KUKA KRL program: MyProgram_060().src

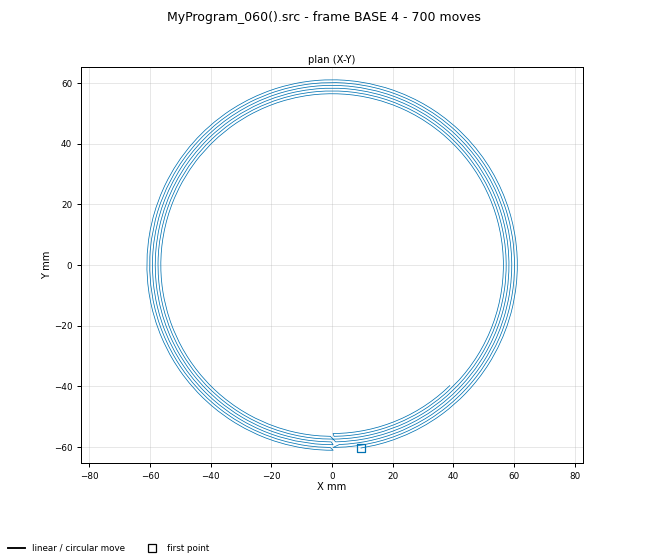
[picture p0: tool path of MyProgram_060().src in frame BASE 4, 700 of 700 moves have a stored position in this frame; points joined in program order, loops and branches not executed]
&ACCESS RVP
&REL 1
&PARAM TEMPLATE = C:\KRC\Roboter\Template\vorgabe
&PARAM EDITMASK = *
DEF MyProgram_060()
; ---- Setting reference (Base) ----
$BASE = BASE_DATA[4]

; --------------------------
; ---- Setting tool (TCP) ----
$TOOL = TOOL_DATA[3]
; --------------------------

$VEL.CP = VEL_APROX_PRINT
Startdeposition()
$VEL.CP = VEL_PRINT
LIN {X 9.5313,Y -60.3261,Z 71,A -85.5574,B 24.8922,C -2.3963,E1 25.0284,E2 529.5228} C_DIS
LIN {X 14.2499,Y -59.3889,Z 71,A -81.7169,B 24.8933,C -2.385,E1 25.0388,E2 525.7139} C_DIS
LIN {X 17.4428,Y -58.5304,Z 71,A -78.0362,B 24.8918,C -2.4016,E1 25.0488,E2 522.0001} C_DIS
LIN {X 20.4744,Y -57.5406,Z 71,A -75.611,B 24.8926,C -2.3923,E1 25.0551,E2 519.6017} C_DIS
LIN {X 24.4545,Y -55.9645,Z 71,A -72.0994,B 24.8931,C -2.3863,E1 25.0642,E2 516.1123} C_DIS
LIN {X 27.8646,Y -54.3472,Z 71,A -68.1205,B 24.8917,C -2.4019,E1 25.0743,E2 512.1067} C_DIS
LIN {X 30.9876,Y -52.6291,Z 71,A -64.3776,B 24.8904,C -2.4171,E1 25.0834,E2 508.339} C_DIS
LIN {X 34.1513,Y -50.6334,Z 71,A -61.0654,B 24.8902,C -2.4192,E1 25.0912,E2 505.0327} C_DIS
LIN {X 36.4572,Y -48.9994,Z 71,A -58.5336,B 24.8899,C -2.4217,E1 25.0969,E2 502.5037} C_DIS
LIN {X 38.3351,Y -47.5447,Z 71,A -55.6589,B 24.8881,C -2.442,E1 25.1032,E2 499.5919} C_DIS
LIN {X 42.1997,Y -44.1508,Z 71,A -51.4902,B 24.8885,C -2.4372,E1 25.1118,E2 495.4512} C_DIS
LIN {X 43.9226,Y -42.4361,Z 71,A -49.1888,B 24.888,C -2.4432,E1 25.1163,E2 493.1454} C_DIS
LIN {X 45.7612,Y -40.4486,Z 71,A -46.6588,B 24.8874,C -2.4493,E1 25.121,E2 490.6124} C_DIS
LIN {X 47.3455,Y -38.5804,Z 71,A -44.3912,B 24.8869,C -2.4545,E1 25.1251,E2 488.3428} C_DIS
LIN {X 49.025,Y -36.4239,Z 71,A -41.5014,B 24.8856,C -2.4692,E1 25.13,E2 485.432} C_DIS
LIN {X 51.0321,Y -33.5526,Z 71,A -38.5025,B 24.8854,C -2.4712,E1 25.1347,E2 482.4432} C_DIS
LIN {X 52.5702,Y -31.0874,Z 71,A -35.4361,B 24.8839,C -2.4873,E1 25.1391,E2 479.3545} C_DIS
LIN {X 54.6001,Y -27.3669,Z 71,A -31.7642,B 24.8835,C -2.4913,E1 25.1439,E2 475.6925} C_DIS
LIN {X 56.3237,Y -23.6157,Z 71,A -27.9982,B 24.8827,C -2.5002,E1 25.1481,E2 471.926} C_DIS
LIN {X 57.7132,Y -19.9822,Z 71,A -23.7879,B 24.8803,C -2.5252,E1 25.1522,E2 467.6801} C_DIS
LIN {X 59.0019,Y -15.7743,Z 71,A -20.3888,B 24.8808,C -2.5199,E1 25.1548,E2 464.3131} C_DIS
LIN {X 59.6127,Y -13.28,Z 71,A -17.5983,B 24.8792,C -2.5369,E1 25.1565,E2 461.4986} C_DIS
LIN {X 60.4839,Y -8.4654,Z 71,A -13.079,B 24.878,C -2.5496,E1 25.1586,E2 456.9758} C_DIS
LIN {X 60.8584,Y -5.1182,Z 71,A -9.9438,B 24.8771,C -2.559,E1 25.1594,E2 453.8369} C_DIS
LIN {X 61.0516,Y -1.6697,Z 71,A -6.9591,B 24.8767,C -2.5628,E1 25.1598,E2 450.8608} C_DIS
LIN {X 61.0519,Y 1.6615,Z 71,A -4.0059,B 24.8762,C -2.5685,E1 25.1597,E2 447.9119} C_DIS
LIN {X 60.9183,Y 4.3667,Z 71,A -0.9984,B 24.8743,C -2.588,E1 25.1591,E2 444.8761} C_DIS
LIN {X 60.5534,Y 7.9589,Z 71,A 2.0459,B 24.8741,C -2.59,E1 25.1582,E2 441.845} C_DIS
LIN {X 60.2672,Y 9.8968,Z 71,A 3.9366,B 24.8734,C -2.597,E1 25.1573,E2 439.9489} C_DIS
LIN {X 59.5946,Y 13.3662,Z 71,A 7.2207,B 24.8725,C -2.6063,E1 25.1554,E2 436.6619} C_DIS
LIN {X 58.852,Y 16.3226,Z 71,A 10.2849,B 24.8711,C -2.62,E1 25.1532,E2 433.5831} C_DIS
LIN {X 57.9096,Y 19.4047,Z 71,A 13.3073,B 24.8702,C -2.6288,E1 25.1506,E2 430.5569} C_DIS
LIN {X 56.5758,Y 23.0049,Z 71,A 16.4909,B 24.8702,C -2.6289,E1 25.1474,E2 427.3908} C_DIS
LIN {X 55.2105,Y 26.1148,Z 71,A 20.5067,B 24.8673,C -2.658,E1 25.1427,E2 423.3278} C_DIS
LIN {X 53.4253,Y 29.5944,Z 71,A 23.4201,B 24.8682,C -2.6495,E1 25.1389,E2 420.4499} C_DIS
LIN {X 51.751,Y 32.4328,Z 71,A 26.9185,B 24.8664,C -2.6673,E1 25.1337,E2 416.9271} C_DIS
LIN {X 49.6974,Y 35.4995,Z 71,A 29.6089,B 24.8674,C -2.6574,E1 25.1295,E2 414.2735} C_DIS
LIN {X 47.4501,Y 38.4518,Z 71,A 33.8937,B 24.8646,C -2.6848,E1 25.122,E2 409.944} C_DIS
LIN {X 44.979,Y 41.3151,Z 71,A 37.3994,B 24.8639,C -2.6916,E1 25.1155,E2 406.4377} C_DIS
LIN {X 42.0159,Y 44.3257,Z 71,A 40.4119,B 24.8654,C -2.6774,E1 25.1096,E2 403.4715} C_DIS
LIN {X 40.4068,Y 45.7971,Z 71,A 42.8829,B 24.864,C -2.6914,E1 25.1044,E2 400.9773} C_DIS
LIN {X 37.3238,Y 48.3424,Z 71,A 46.173,B 24.8644,C -2.6875,E1 25.0973,E2 397.7088} C_DIS
LIN {X 34.8357,Y 50.1649,Z 71,A 49.3042,B 24.8633,C -2.6979,E1 25.0902,E2 394.564} C_DIS
LIN {X 32.4004,Y 51.7711,Z 71,A 52.3355,B 24.8622,C -2.7089,E1 25.0831,E2 391.5166} C_DIS
LIN {X 30.0717,Y 53.1588,Z 71,A 54.7481,B 24.8622,C -2.7094,E1 25.0773,E2 389.1099} C_DIS
LIN {X 27.325,Y 54.6209,Z 71,A 57.7015,B 24.8617,C -2.7139,E1 25.0699,E2 386.154} C_DIS
LIN {X 23.8442,Y 56.2274,Z 71,A 61.6491,B 24.8605,C -2.7258,E1 25.0598,E2 382.1879} C_DIS
LIN {X 20.335,Y 57.5895,Z 71,A 64.8251,B 24.8609,C -2.7211,E1 25.0515,E2 379.0299} C_DIS
LIN {X 17.5465,Y 58.4996,Z 71,A 67.5039,B 24.8609,C -2.7215,E1 25.0444,E2 376.3549} C_DIS
LIN {X 12.2273,Y 59.8376,Z 71,A 72.4673,B 24.861,C -2.7203,E1 25.031,E2 371.4014} C_DIS
LIN {X 7.8287,Y 60.5703,Z 71,A 76.8844,B 24.8604,C -2.7266,E1 25.0187,E2 366.9737} C_DIS
LIN {X 4.1966,Y 60.9298,Z 71,A 80.4406,B 24.8601,C -2.7296,E1 25.0088,E2 363.4121} C_DIS
LIN {X 1.5588,Y 61.055,Z 71,A 83.8521,B 24.858,C -2.7493,E1 24.9992,E2 359.9544} C_DIS
LIN {X -2.3408,Y 61.0299,Z 71,A 86.0215,B 24.8614,C -2.7168,E1 24.9933,E2 357.8622} C_DIS
LIN {X -4.5003,Y 60.9082,Z 71,A 88.4038,B 24.8607,C -2.7234,E1 24.9866,E2 355.4635} C_DIS
LIN {X -7.1884,Y 60.6497,Z 71,A 90.9106,B 24.8609,C -2.7215,E1 24.9797,E2 352.9596} C_DIS
LIN {X -9.8136,Y 60.2811,Z 71,A 93.7308,B 24.8604,C -2.7267,E1 24.9719,E2 350.1247} C_DIS
LIN {X -12.1519,Y 59.8531,Z 71,A 96.1882,B 24.8601,C -2.7295,E1 24.9651,E2 347.6576} C_DIS
LIN {X -16.0091,Y 58.9386,Z 71,A 99.3972,B 24.8615,C -2.7155,E1 24.9565,E2 344.4773} C_DIS
LIN {X -18.5062,Y 58.203,Z 71,A 101.8781,B 24.8617,C -2.7136,E1 24.9499,E2 341.9967} C_DIS
LIN {X -21.2409,Y 57.2618,Z 71,A 104.8189,B 24.8616,C -2.7148,E1 24.9421,E2 339.0473} C_DIS
LIN {X -24.891,Y 55.7722,Z 71,A 108.3276,B 24.8625,C -2.7058,E1 24.9332,E2 335.5519} C_DIS
LIN {X -27.9296,Y 54.314,Z 71,A 111.689,B 24.8626,C -2.7047,E1 24.9247,E2 332.1842} C_DIS
LIN {X -31.0887,Y 52.5694,Z 71,A 114.4199,B 24.8645,C -2.6861,E1 24.9182,E2 329.4896} C_DIS
LIN {X -33.5476,Y 51.0353,Z 71,A 117.4155,B 24.8645,C -2.6864,E1 24.9111,E2 326.4838} C_DIS
LIN {X -35.2032,Y 49.9088,Z 71,A 119.7238,B 24.864,C -2.691,E1 24.9058,E2 324.1566} C_DIS
LIN {X -38.7067,Y 47.2435,Z 71,A 123.6795,B 24.8652,C -2.679,E1 24.8971,E2 320.2151} C_DIS
LIN {X -41.8199,Y 44.5094,Z 71,A 127.6927,B 24.8659,C -2.6726,E1 24.8888,E2 316.201} C_DIS
LIN {X -44.4407,Y 41.8923,Z 71,A 131.5933,B 24.8659,C -2.6723,E1 24.8812,E2 312.2843} C_DIS
LIN {X -47.0833,Y 38.9004,Z 71,A 135.1961,B 24.8671,C -2.6601,E1 24.8747,E2 308.6942} C_DIS
LIN {X -49.9457,Y 35.1511,Z 71,A 138.9483,B 24.8695,C -2.6358,E1 24.8685,E2 304.9819} C_DIS
LIN {X -52.1565,Y 31.7765,Z 71,A 142.9291,B 24.8702,C -2.629,E1 24.8625,E2 300.9973} C_DIS
LIN {X -54.0948,Y 28.3504,Z 71,A 146.6636,B 24.8712,C -2.6192,E1 24.8575,E2 297.2666} C_DIS
LIN {X -55.2292,Y 26.0746,Z 71,A 148.9802,B 24.872,C -2.6109,E1 24.8546,E2 294.9573} C_DIS
LIN {X -56.5378,Y 23.0984,Z 71,A 152.6229,B 24.8718,C -2.6127,E1 24.8506,E2 291.2902} C_DIS
LIN {X -58.0535,Y 18.9702,Z 71,A 156.411,B 24.8737,C -2.594,E1 24.8472,E2 287.5253} C_DIS
LIN {X -59.019,Y 15.7117,Z 71,A 159.9204,B 24.8741,C -2.59,E1 24.8445,E2 284.0052} C_DIS
LIN {X -59.9673,Y 11.5748,Z 71,A 164.0224,B 24.8751,C -2.5797,E1 24.8421,E2 279.9035} C_DIS
LIN {X -60.5089,Y 8.2947,Z 71,A 166.6181,B 24.8769,C -2.5603,E1 24.8411,E2 277.3386} C_DIS
LIN {X -60.9649,Y 3.6625,Z 71,A 170.8735,B 24.8785,C -2.5445,E1 24.84,E2 273.0955} C_DIS
LIN {X -61.0554,Y -1.5469,Z 71,A 176.0124,B 24.8795,C -2.5336,E1 24.8399,E2 267.9518} C_DIS
LIN {X -60.7658,Y -6.133,Z 71,A -179.9583,B 24.8813,C -2.5149,E1 24.8407,E2 263.9428} C_DIS
LIN {X -60.3491,Y -9.3826,Z 71,A -175.9941,B 24.8806,C -2.5217,E1 24.8422,E2 259.9388} C_DIS
LIN {X -59.747,Y -12.6645,Z 71,A -173.4662,B 24.8826,C -2.5011,E1 24.8436,E2 257.4453} C_DIS
LIN {X -59.1871,Y -15.065,Z 71,A -170.4431,B 24.882,C -2.5072,E1 24.8456,E2 254.3899} C_DIS
LIN {X -58.0142,Y -19.0915,Z 71,A -166.5799,B 24.8832,C -2.4943,E1 24.8489,E2 250.5354} C_DIS
LIN {X -56.7141,Y -22.6646,Z 71,A -163.1855,B 24.8845,C -2.4808,E1 24.8523,E2 247.1541} C_DIS
LIN {X -55.5425,Y -25.4007,Z 71,A -160.3729,B 24.8852,C -2.4734,E1 24.8555,E2 244.3438} C_DIS
LIN {X -53.531,Y -29.4038,Z 71,A -156.4605,B 24.8867,C -2.4566,E1 24.8605,E2 240.4507} C_DIS
LIN {X -52.1052,Y -31.8609,Z 71,A -153.6626,B 24.8871,C -2.4522,E1 24.8645,E2 237.6489} C_DIS
LIN {X -50.2298,Y -34.7424,Z 71,A -150.4202,B 24.8879,C -2.4444,E1 24.8695,E2 234.4088} C_DIS
LIN {X -49.0978,Y -36.3255,Z 71,A -147.7959,B 24.8869,C -2.4553,E1 24.874,E2 231.7457} C_DIS
LIN {X -47.1038,Y -38.8757,Z 71,A -145.7362,B 24.8892,C -2.4295,E1 24.8775,E2 229.7381} C_DIS
LIN {X -44.3514,Y -41.9886,Z 71,A -141.8795,B 24.8901,C -2.4201,E1 24.8847,E2 225.8867} C_DIS
LIN {X -42.4737,Y -43.8866,Z 71,A -139.3874,B 24.8906,C -2.4147,E1 24.8896,E2 223.3971} C_DIS
LIN {X -40.1119,Y -46.0553,Z 71,A -136.1393,B 24.8906,C -2.4135,E1 24.8964,E2 220.1388} C_DIS
LIN {X -37.6052,Y -48.1241,Z 71,A -132.9342,B 24.8909,C -2.411,E1 24.9033,E2 216.9274} C_DIS
LIN {X -34.1663,Y -50.6233,Z 71,A -129.0128,B 24.8916,C -2.4032,E1 24.9123,E2 213.0113} C_DIS
LIN {X -31.9807,Y -52.0325,Z 71,A -126.2783,B 24.8914,C -2.4055,E1 24.9188,E2 210.2627} C_DIS
LIN {X -28.8608,Y -53.8255,Z 71,A -122.7562,B 24.8915,C -2.404,E1 24.9274,E2 206.7341} C_DIS
LIN {X -24.5436,Y -55.9257,Z 71,A -118.7195,B 24.8929,C -2.3893,E1 24.9376,E2 202.7222} C_DIS
LIN {X -21.8949,Y -57.0142,Z 71,A -116.0165,B 24.8931,C -2.3871,E1 24.9446,E2 200.0187} C_DIS
LIN {X -19.0924,Y -58.014,Z 71,A -112.065,B 24.8911,C -2.4093,E1 24.9552,E2 196.007} C_DIS
LIN {X -15.3082,Y -59.1246,Z 71,A -110.0337,B 24.8944,C -2.3718,E1 24.9605,E2 194.0618} C_DIS
LIN {X -11.3347,Y -60.0135,Z 71,A -105.6294,B 24.8935,C -2.3823,E1 24.9726,E2 189.6269} C_DIS
LIN {X -8.9195,Y -60.4202,Z 71,A -102.8059,B 24.8925,C -2.3931,E1 24.9804,E2 186.7755} C_DIS
LIN {X -5.3261,Y -60.8421,Z 71,A -100.1582,B 24.894,C -2.3766,E1 24.9877,E2 184.1654} C_DIS
LIN {X -1.8193,Y -61.047,Z 71,A -96.6621,B 24.8936,C -2.3812,E1 24.9975,E2 180.6574} C_DIS
LIN {X 0.3504,Y -61.0663,Z 71,A -94.3682,B 24.893,C -2.3875,E1 25.0039,E2 178.3488} C_DIS
Enddeposition()
LIN {X 0.3504,Y -61.0663,Z 71,A -94.3682,B 24.893,C -2.3875,E1 25.0039,E2 178.3488} C_DIS
Startdeposition()
$VEL.CP = VEL_PRINT
LIN {X -0.6024,Y -60.1527,Z 71,A -97.3329,B 24.8956,C -2.3591,E1 24.9955,E2 181.381} C_DIS
LIN {X -4.5861,Y -59.9805,Z 71,A -100.7162,B 24.8948,C -2.3675,E1 24.9861,E2 184.7453} C_DIS
LIN {X -7.8091,Y -59.6461,Z 71,A -103.721,B 24.8946,C -2.3697,E1 24.9777,E2 187.747} C_DIS
LIN {X -10.2074,Y -59.2836,Z 71,A -106.4784,B 24.8954,C -2.3612,E1 24.9701,E2 190.5271} C_DIS
LIN {X -14.9728,Y -58.262,Z 71,A -111.6213,B 24.8961,C -2.3536,E1 24.9561,E2 195.6951} C_DIS
LIN {X -18.2838,Y -57.3098,Z 71,A -114.2777,B 24.8948,C -2.3683,E1 24.9491,E2 198.3211} C_DIS
LIN {X -22.1363,Y -55.9344,Z 71,A -118.2942,B 24.8946,C -2.3695,E1 24.9385,E2 202.3432} C_DIS
LIN {X -25.8621,Y -54.3125,Z 71,A -121.9851,B 24.894,C -2.3773,E1 24.9292,E2 206.0246} C_DIS
LIN {X -28.523,Y -52.9634,Z 71,A -124.9156,B 24.8938,C -2.3791,E1 24.9219,E2 208.9587} C_DIS
LIN {X -32.2792,Y -50.7619,Z 71,A -128.3777,B 24.8921,C -2.3983,E1 24.9137,E2 212.3858} C_DIS
LIN {X -35.6023,Y -48.4885,Z 71,A -132.4546,B 24.8919,C -2.3999,E1 24.9044,E2 216.4728} C_DIS
LIN {X -37.3846,Y -47.128,Z 71,A -134.7657,B 24.8919,C -2.4003,E1 24.8993,E2 218.7913} C_DIS
LIN {X -39.1876,Y -45.6403,Z 71,A -137.4375,B 24.8923,C -2.3961,E1 24.8935,E2 221.4834} C_DIS
LIN {X -41.213,Y -43.8194,Z 71,A -139.9645,B 24.8917,C -2.4025,E1 24.8884,E2 224.0055} C_DIS
LIN {X -43.7788,Y -41.2562,Z 71,A -143.9978,B 24.892,C -2.3993,E1 24.8805,E2 228.064} C_DIS
LIN {X -46.0507,Y -38.7051,Z 71,A -146.008,B 24.8892,C -2.4293,E1 24.877,E2 230.0116} C_DIS
LIN {X -48.4635,Y -35.6364,Z 71,A -150.0555,B 24.889,C -2.4321,E1 24.8701,E2 234.0718} C_DIS
LIN {X -50.0061,Y -33.4377,Z 71,A -152.5742,B 24.8883,C -2.4391,E1 24.8661,E2 236.5861} C_DIS
LIN {X -51.3259,Y -31.374,Z 71,A -155.0698,B 24.8881,C -2.4421,E1 24.8624,E2 239.0872} C_DIS
LIN {X -52.4055,Y -29.5358,Z 71,A -156.947,B 24.8873,C -2.4502,E1 24.8598,E2 240.9548} C_DIS
LIN {X -53.8809,Y -26.7487,Z 71,A -160.2346,B 24.887,C -2.4533,E1 24.8556,E2 244.2528} C_DIS
LIN {X -55.2221,Y -23.8581,Z 71,A -163.2733,B 24.8863,C -2.4617,E1 24.8521,E2 247.288} C_DIS
LIN {X -56.306,Y -21.1733,Z 71,A -166.1679,B 24.8858,C -2.4672,E1 24.8492,E2 250.1857} C_DIS
LIN {X -57.2806,Y -18.3741,Z 71,A -168.5005,B 24.8842,C -2.4841,E1 24.8471,E2 252.4913} C_DIS
LIN {X -58.3236,Y -14.7331,Z 71,A -171.8693,B 24.8828,C -2.499,E1 24.8446,E2 255.8439} C_DIS
LIN {X -59.0185,Y -11.6424,Z 71,A -175.8143,B 24.8834,C -2.492,E1 24.8423,E2 259.8291} C_DIS
LIN {X -59.7898,Y -6.6302,Z 71,A 179.6959,B 24.8815,C -2.5128,E1 24.8406,E2 264.2958} C_DIS
LIN {X -60.1279,Y -1.812,Z 71,A 175.3491,B 24.8797,C -2.5317,E1 24.8398,E2 268.6237} C_DIS
LIN {X -60.0961,Y 2.6668,Z 71,A 171.1828,B 24.8782,C -2.5469,E1 24.84,E2 272.7787} C_DIS
LIN {X -59.9771,Y 4.6287,Z 71,A 168.4056,B 24.8792,C -2.5371,E1 24.8405,E2 275.5959} C_DIS
LIN {X -59.5679,Y 8.3859,Z 71,A 164.4883,B 24.8786,C -2.543,E1 24.842,E2 279.5225} C_DIS
LIN {X -58.2854,Y 14.882,Z 71,A 159.1838,B 24.875,C -2.5801,E1 24.845,E2 284.7697} C_DIS
LIN {X -57.5897,Y 17.3797,Z 71,A 156.2187,B 24.8751,C -2.5791,E1 24.8474,E2 287.7543} C_DIS
LIN {X -56.6004,Y 20.3742,Z 71,A 152.7791,B 24.875,C -2.5807,E1 24.8506,E2 291.2096} C_DIS
LIN {X -54.5804,Y 25.2911,Z 71,A 147.6942,B 24.8735,C -2.5954,E1 24.8562,E2 296.2874} C_DIS
LIN {X -52.0908,Y 30.0868,Z 71,A 142.7359,B 24.8718,C -2.6134,E1 24.8628,E2 301.2288} C_DIS
LIN {X -50.0697,Y 33.3421,Z 71,A 139.4301,B 24.8702,C -2.6295,E1 24.8678,E2 304.5128} C_DIS
LIN {X -47.9265,Y 36.3542,Z 71,A 135.292,B 24.8703,C -2.628,E1 24.8747,E2 308.6745} C_DIS
LIN {X -45.189,Y 39.7069,Z 71,A 131.43,B 24.8688,C -2.643,E1 24.8816,E2 312.5182} C_DIS
LIN {X -42.5715,Y 42.502,Z 71,A 127.6514,B 24.8682,C -2.6494,E1 24.889,E2 316.2978} C_DIS
LIN {X -38.7988,Y 45.9716,Z 71,A 123.5322,B 24.8657,C -2.6743,E1 24.8975,E2 320.3741} C_DIS
LIN {X -36.4037,Y 47.8889,Z 71,A 119.9369,B 24.8663,C -2.6681,E1 24.9054,E2 323.9974} C_DIS
LIN {X -33.3449,Y 50.0673,Z 71,A 116.4337,B 24.8655,C -2.6764,E1 24.9135,E2 327.4926} C_DIS
LIN {X -30.3333,Y 51.9485,Z 71,A 112.1211,B 24.8666,C -2.6653,E1 24.9239,E2 331.8448} C_DIS
LIN {X -26.9443,Y 53.7838,Z 71,A 109.5322,B 24.864,C -2.6913,E1 24.9302,E2 334.3787} C_DIS
LIN {X -25.1235,Y 54.6584,Z 71,A 107.0936,B 24.8647,C -2.6845,E1 24.9365,E2 336.8395} C_DIS
LIN {X -20.6035,Y 56.5168,Z 71,A 103.1848,B 24.8626,C -2.705,E1 24.9465,E2 340.7081} C_DIS
LIN {X -18.7117,Y 57.1712,Z 71,A 100.3683,B 24.8641,C -2.6897,E1 24.9541,E2 343.5661} C_DIS
LIN {X -15.3925,Y 58.1534,Z 71,A 96.9099,B 24.8641,C -2.6899,E1 24.9634,E2 347.0292} C_DIS
LIN {X -12.2651,Y 58.8918,Z 71,A 94.9035,B 24.8618,C -2.7131,E1 24.9687,E2 348.9829} C_DIS
LIN {X -8.8298,Y 59.5035,Z 71,A 91.5704,B 24.8615,C -2.7153,E1 24.9779,E2 352.314} C_DIS
LIN {X -6.9747,Y 59.7495,Z 71,A 89.4695,B 24.8621,C -2.71,E1 24.9838,E2 354.4291} C_DIS
LIN {X -3.534,Y 60.0517,Z 71,A 86.5713,B 24.8611,C -2.7193,E1 24.9918,E2 357.3064} C_DIS
LIN {X 1.304,Y 60.1414,Z 71,A 82.0334,B 24.8609,C -2.7218,E1 25.0045,E2 361.8384} C_DIS
LIN {X 4.0722,Y 60.0172,Z 71,A 78.6283,B 24.8625,C -2.7062,E1 25.014,E2 365.2794} C_DIS
LIN {X 7.8042,Y 59.6465,Z 71,A 75.1627,B 24.8623,C -2.7077,E1 25.0236,E2 368.7387} C_DIS
LIN {X 12.0069,Y 58.9448,Z 71,A 70.4446,B 24.8639,C -2.6925,E1 25.0366,E2 373.4877} C_DIS
LIN {X 15.4197,Y 58.146,Z 71,A 67.8014,B 24.8626,C -2.705,E1 25.0437,E2 376.097} C_DIS
LIN {X 19.1131,Y 57.0381,Z 71,A 64.5218,B 24.862,C -2.7106,E1 25.0524,E2 379.3574} C_DIS
LIN {X 21.3935,Y 56.2226,Z 71,A 61.8822,B 24.863,C -2.7014,E1 25.0593,E2 382.0134} C_DIS
LIN {X 24.6497,Y 54.873,Z 71,A 58.9077,B 24.8625,C -2.7061,E1 25.0669,E2 384.9696} C_DIS
LIN {X 27.2605,Y 53.624,Z 71,A 55.6988,B 24.8638,C -2.6929,E1 25.075,E2 388.2013} C_DIS
LIN {X 29.7238,Y 52.2994,Z 71,A 53.3009,B 24.8636,C -2.695,E1 25.0808,E2 390.587} C_DIS
LIN {X 33.2527,Y 50.1292,Z 71,A 49.2867,B 24.8644,C -2.6875,E1 25.0903,E2 394.606} C_DIS
LIN {X 36.2291,Y 48.022,Z 71,A 46.3877,B 24.8637,C -2.6945,E1 25.0968,E2 397.4782} C_DIS
LIN {X 38.8634,Y 45.9165,Z 71,A 42.5979,B 24.8656,C -2.6756,E1 25.1051,E2 401.2986} C_DIS
LIN {X 40.7623,Y 44.2392,Z 71,A 40.4405,B 24.8655,C -2.6767,E1 25.1096,E2 403.4448} C_DIS
LIN {X 43.3467,Y 41.7099,Z 71,A 36.8774,B 24.8665,C -2.6668,E1 25.1166,E2 407.0163} C_DIS
LIN {X 44.7731,Y 40.1749,Z 71,A 34.1484,B 24.8686,C -2.6457,E1 25.1218,E2 409.783} C_DIS
LIN {X 48.2371,Y 35.9425,Z 71,A 29.7537,B 24.8679,C -2.6521,E1 25.1293,E2 414.142} C_DIS
LIN {X 50.1978,Y 33.1486,Z 71,A 26.3954,B 24.869,C -2.6415,E1 25.1346,E2 417.5087} C_DIS
LIN {X 51.4362,Y 31.1925,Z 71,A 24.2678,B 24.8694,C -2.6376,E1 25.1377,E2 419.6348} C_DIS
LIN {X 52.9238,Y 28.5959,Z 71,A 21.7482,B 24.8694,C -2.6377,E1 25.1411,E2 422.1409} C_DIS
LIN {X 54.4607,Y 25.5483,Z 71,A 18.7154,B 24.8697,C -2.634,E1 25.1449,E2 425.1664} C_DIS
LIN {X 55.7019,Y 22.7144,Z 71,A 14.5086,B 24.8735,C -2.5961,E1 25.1495,E2 429.4397} C_DIS
LIN {X 56.8361,Y 19.7069,Z 71,A 12.565,B 24.8718,C -2.6135,E1 25.1513,E2 431.3313} C_DIS
LIN {X 57.558,Y 17.4882,Z 71,A 9.0058,B 24.8755,C -2.5754,E1 25.1543,E2 434.9602} C_DIS
LIN {X 58.5266,Y 13.9009,Z 71,A 6.6587,B 24.8738,C -2.5928,E1 25.1558,E2 437.2525} C_DIS
LIN {X 59.4677,Y 9.0697,Z 71,A 2.1525,B 24.8748,C -2.5828,E1 25.1581,E2 441.7561} C_DIS
LIN {X 59.7772,Y 6.7379,Z 71,A -0.8146,B 24.8771,C -2.5585,E1 25.1591,E2 444.7632} C_DIS
LIN {X 60.1241,Y 1.9359,Z 71,A -5.3772,B 24.8784,C -2.5447,E1 25.1598,E2 449.3313} C_DIS
LIN {X 60.1423,Y -1.2551,Z 71,A -7.9162,B 24.8782,C -2.547,E1 25.1597,E2 451.8497} C_DIS
LIN {X 59.9587,Y -4.8584,Z 71,A -11.4456,B 24.8795,C -2.5339,E1 25.1591,E2 455.3892} C_DIS
LIN {X 59.6595,Y -7.707,Z 71,A -13.9397,B 24.8798,C -2.5309,E1 25.1583,E2 457.8756} C_DIS
LIN {X 59.1993,Y -10.6817,Z 71,A -16.9157,B 24.8809,C -2.5192,E1 25.1569,E2 460.8617} C_DIS
LIN {X 58.41,Y -14.3854,Z 71,A -20.7632,B 24.8825,C -2.5022,E1 25.1545,E2 464.7271} C_DIS
LIN {X 57.5402,Y -17.5459,Z 71,A -23.9267,B 24.8835,C -2.4915,E1 25.152,E2 467.8977} C_DIS
LIN {X 56.1297,Y -21.6368,Z 71,A -27.5493,B 24.8835,C -2.4909,E1 25.1486,E2 471.5016} C_DIS
LIN {X 55.2437,Y -23.8085,Z 71,A -29.912,B 24.8845,C -2.4811,E1 25.146,E2 473.8744} C_DIS
LIN {X 53.949,Y -26.6115,Z 71,A -32.8209,B 24.8852,C -2.4732,E1 25.1425,E2 476.7863} C_DIS
LIN {X 51.7218,Y -30.7168,Z 71,A -36.5119,B 24.8847,C -2.4785,E1 25.1376,E2 480.4456} C_DIS
LIN {X 49.2068,Y -34.6039,Z 71,A -41.5992,B 24.8873,C -2.4502,E1 25.1298,E2 485.5744} C_DIS
LIN {X 47.3592,Y -37.0921,Z 71,A -44.6534,B 24.8883,C -2.4399,E1 25.1246,E2 488.6382} C_DIS
LIN {X 45.7436,Y -39.0663,Z 71,A -46.7003,B 24.888,C -2.4427,E1 25.1209,E2 490.6693} C_DIS
LIN {X 44.4188,Y -40.5665,Z 71,A -48.6586,B 24.8886,C -2.4367,E1 25.1173,E2 492.6331} C_DIS
LIN {X 42.6589,Y -42.4135,Z 71,A -51.3079,B 24.8896,C -2.4257,E1 25.1121,E2 495.297} C_DIS
LIN {X 40.0318,Y -44.9012,Z 71,A -54.5017,B 24.8898,C -2.4236,E1 25.1056,E2 498.4828} C_DIS
LIN {X 37.682,Y -46.8912,Z 71,A -57.3654,B 24.8902,C -2.4187,E1 25.0994,E2 501.347} C_DIS
LIN {X 36.2809,Y -47.9831,Z 71,A -59.4249,B 24.8913,C -2.4067,E1 25.0948,E2 503.4273} C_DIS
LIN {X 33.4816,Y -49.9772,Z 71,A -62.5144,B 24.8915,C -2.4044,E1 25.0877,E2 506.5117} C_DIS
LIN {X 30.9995,Y -51.5535,Z 71,A -65.451,B 24.8923,C -2.3961,E1 25.0807,E2 509.4587} C_DIS
LIN {X 28.3987,Y -53.0308,Z 71,A -68.5489,B 24.8932,C -2.3856,E1 25.0731,E2 512.5725} C_DIS
LIN {X 25.2337,Y -54.6071,Z 71,A -71.4802,B 24.8928,C -2.3901,E1 25.0658,E2 515.4855} C_DIS
LIN {X 22.8346,Y -55.653,Z 71,A -73.9642,B 24.8931,C -2.3867,E1 25.0594,E2 517.9717} C_DIS
LIN {X 20.2552,Y -56.6435,Z 71,A -76.6449,B 24.8935,C -2.3821,E1 25.0523,E2 520.6575} C_DIS
LIN {X 17.1851,Y -57.6483,Z 71,A -79.9352,B 24.8943,C -2.3739,E1 25.0435,E2 523.9614} C_DIS
LIN {X 14.4605,Y -58.3917,Z 71,A -82.1861,B 24.8936,C -2.3808,E1 25.0375,E2 526.1925} C_DIS
LIN {X 10.6878,Y -59.1982,Z 71,A -85.6372,B 24.8935,C -2.3824,E1 25.0281,E2 529.6353} C_DIS
LIN {X 8.7278,Y -59.5193,Z 71,A -89.2244,B 24.8968,C -2.3449,E1 25.018,E2 533.3083} C_DIS
LIN {X 4.5328,Y -59.9848,Z 71,A -92.1184,B 24.8949,C -2.3666,E1 25.0101,E2 536.1492} C_DIS
LIN {X 0.3297,Y -60.1458,Z 71,A -94.3994,B 24.8917,C -2.4023,E1 25.004,E2 538.3448} C_DIS
Enddeposition()
LIN {X 0.3297,Y -60.1458,Z 71,A -94.3994,B 24.8917,C -2.4023,E1 25.004,E2 538.3448} C_DIS
Startdeposition()
$VEL.CP = VEL_PRINT
LIN {X 2.3476,Y -59.1901,Z 71,A -92.6158,B 24.8906,C -2.4149,E1 25.009,E2 536.5318} C_DIS
LIN {X 5.1105,Y -59.0155,Z 71,A -89.1553,B 24.8889,C -2.4331,E1 25.0187,E2 533.0299} C_DIS
LIN {X 8.5308,Y -58.6192,Z 71,A -86.7615,B 24.8906,C -2.4149,E1 25.0252,E2 530.6814} C_DIS
LIN {X 10.9463,Y -58.2167,Z 71,A -84.5732,B 24.8907,C -2.4128,E1 25.0312,E2 528.5004} C_DIS
LIN {X 12.903,Y -57.8147,Z 71,A -82.4491,B 24.8902,C -2.4188,E1 25.037,E2 526.3651} C_DIS
LIN {X 15.513,Y -57.169,Z 71,A -79.8384,B 24.8899,C -2.4216,E1 25.0441,E2 523.7516} C_DIS
LIN {X 18.3053,Y -56.3371,Z 71,A -76.8889,B 24.8894,C -2.4278,E1 25.052,E2 520.7927} C_DIS
LIN {X 21.8293,Y -55.0678,Z 71,A -73.7259,B 24.8899,C -2.4223,E1 25.0602,E2 517.6495} C_DIS
LIN {X 23.4437,Y -54.4004,Z 71,A -71.2991,B 24.8881,C -2.4414,E1 25.0665,E2 515.1833} C_DIS
LIN {X 27.932,Y -52.2383,Z 71,A -67.1599,B 24.8888,C -2.4337,E1 25.0768,E2 511.0734} C_DIS
LIN {X 30.5511,Y -50.7507,Z 71,A -63.7965,B 24.8874,C -2.4492,E1 25.085,E2 507.6836} C_DIS
LIN {X 32.8108,Y -49.3199,Z 71,A -61.176,B 24.8869,C -2.455,E1 25.0911,E2 505.0582} C_DIS
LIN {X 36.1038,Y -46.9623,Z 71,A -57.7367,B 24.8872,C -2.452,E1 25.0988,E2 501.6382} C_DIS
LIN {X 38.0627,Y -45.3895,Z 71,A -54.7261,B 24.8854,C -2.4708,E1 25.1053,E2 498.5946} C_DIS
LIN {X 40.9142,Y -42.8374,Z 71,A -51.2565,B 24.8851,C -2.4739,E1 25.1124,E2 495.1317} C_DIS
LIN {X 43.5568,Y -40.1468,Z 71,A -47.873,B 24.8849,C -2.4766,E1 25.1189,E2 491.7565} C_DIS
LIN {X 45.297,Y -38.172,Z 71,A -45.0831,B 24.8837,C -2.4889,E1 25.124,E2 488.9502} C_DIS
LIN {X 47.7459,Y -35.0611,Z 71,A -41.788,B 24.884,C -2.4863,E1 25.1296,E2 485.6768} C_DIS
LIN {X 49.4078,Y -32.6776,Z 71,A -38.2296,B 24.8816,C -2.5118,E1 25.1352,E2 482.0757} C_DIS
LIN {X 50.999,Y -30.1338,Z 71,A -35.3369,B 24.8808,C -2.5198,E1 25.1394,E2 479.1789} C_DIS
LIN {X 53.2383,Y -25.9758,Z 71,A -31.4083,B 24.881,C -2.5177,E1 25.1444,E2 475.2761} C_DIS
LIN {X 54.1566,Y -24.0026,Z 71,A -29.0597,B 24.8799,C -2.5298,E1 25.1471,E2 472.9116} C_DIS
LIN {X 55.3963,Y -20.9808,Z 71,A -25.9604,B 24.8791,C -2.5379,E1 25.1503,E2 469.8104} C_DIS
LIN {X 56.5244,Y -17.7192,Z 71,A -22.9217,B 24.8788,C -2.541,E1 25.1529,E2 466.7817} C_DIS
LIN {X 57.1128,Y -15.721,Z 71,A -20.2553,B 24.8767,C -2.5629,E1 25.1549,E2 464.0787} C_DIS
LIN {X 58.027,Y -11.9084,Z 71,A -16.941,B 24.8767,C -2.5632,E1 25.1569,E2 460.7828} C_DIS
LIN {X 58.4563,Y -9.5834,Z 71,A -13.9915,B 24.8744,C -2.5865,E1 25.1583,E2 457.7957} C_DIS
LIN {X 58.95,Y -5.8274,Z 71,A -11.2766,B 24.8755,C -2.5751,E1 25.1591,E2 455.1237} C_DIS
LIN {X 59.1986,Y -2.139,Z 71,A -7.8773,B 24.8748,C -2.5821,E1 25.1597,E2 451.728} C_DIS
LIN {X 59.236,Y 0.3962,Z 71,A -4.9045,B 24.8728,C -2.6024,E1 25.1597,E2 448.725} C_DIS
LIN {X 59.1318,Y 3.5268,Z 71,A -1.8651,B 24.8719,C -2.6122,E1 25.1593,E2 445.6806} C_DIS
LIN {X 58.793,Y 7.2422,Z 71,A 1.3669,B 24.8717,C -2.6144,E1 25.1584,E2 442.4625} C_DIS
LIN {X 58.1653,Y 11.2122,Z 71,A 5.6129,B 24.8696,C -2.6349,E1 25.1564,E2 438.1928} C_DIS
LIN {X 56.8339,Y 16.6994,Z 71,A 10.826,B 24.8686,C -2.6453,E1 25.1527,E2 432.9851} C_DIS
LIN {X 55.949,Y 19.4597,Z 71,A 13.1443,B 24.8689,C -2.642,E1 25.1507,E2 430.6877} C_DIS
LIN {X 54.8281,Y 22.4239,Z 71,A 16.9515,B 24.8663,C -2.6684,E1 25.1468,E2 426.8393} C_DIS
LIN {X 53.7108,Y 24.9818,Z 71,A 19.631,B 24.8656,C -2.6754,E1 25.1437,E2 424.1577} C_DIS
LIN {X 52.1824,Y 28.0357,Z 71,A 23.0907,B 24.8643,C -2.688,E1 25.1392,E2 420.6865} C_DIS
LIN {X 50.4302,Y 31.0785,Z 71,A 25.7008,B 24.8653,C -2.6784,E1 25.1355,E2 418.1125} C_DIS
LIN {X 49.1678,Y 33.0381,Z 71,A 28.1942,B 24.8641,C -2.6897,E1 25.1317,E2 415.6049} C_DIS
LIN {X 47.8309,Y 34.945,Z 71,A 30.2471,B 24.8641,C -2.6906,E1 25.1283,E2 413.5599} C_DIS
LIN {X 46.0521,Y 37.2579,Z 71,A 34.2412,B 24.8606,C -2.7244,E1 25.1213,E2 409.5042} C_DIS
LIN {X 43.7248,Y 39.9637,Z 71,A 36.1479,B 24.8635,C -2.6964,E1 25.1179,E2 407.6723} C_DIS
LIN {X 41.0683,Y 42.6889,Z 71,A 40.3497,B 24.8615,C -2.716,E1 25.1096,E2 403.4421} C_DIS
LIN {X 39.5214,Y 44.1248,Z 71,A 42.387,B 24.8611,C -2.7199,E1 25.1053,E2 401.4037} C_DIS
LIN {X 35.8359,Y 47.1682,Z 71,A 47.1853,B 24.8598,C -2.7322,E1 25.0949,E2 396.5942} C_DIS
LIN {X 33.4449,Y 48.8924,Z 71,A 49.6948,B 24.8601,C -2.7293,E1 25.0892,E2 394.1003} C_DIS
LIN {X 31.1857,Y 50.3626,Z 71,A 52.7536,B 24.8587,C -2.7433,E1 25.0819,E2 391.0182} C_DIS
LIN {X 27.1929,Y 52.6258,Z 71,A 57.1352,B 24.8582,C -2.7479,E1 25.0711,E2 386.6382} C_DIS
LIN {X 24.0879,Y 54.1175,Z 71,A 60.3526,B 24.858,C -2.7492,E1 25.063,E2 383.4259} C_DIS
LIN {X 21.0939,Y 55.3535,Z 71,A 63.5113,B 24.8577,C -2.7528,E1 25.0548,E2 380.2657} C_DIS
LIN {X 18.1782,Y 56.3782,Z 71,A 66.1842,B 24.8581,C -2.7485,E1 25.0477,E2 377.6083} C_DIS
LIN {X 14.6477,Y 57.3968,Z 71,A 70.5126,B 24.8562,C -2.7673,E1 25.036,E2 373.2421} C_DIS
LIN {X 9.3742,Y 58.4908,Z 71,A 75.6357,B 24.8562,C -2.7673,E1 25.0219,E2 368.1245} C_DIS
LIN {X 5.4181,Y 58.988,Z 71,A 79.8154,B 24.8554,C -2.7746,E1 25.0103,E2 363.9302} C_DIS
LIN {X 2.0213,Y 59.2022,Z 71,A 81.9515,B 24.8579,C -2.7505,E1 25.0045,E2 361.8522} C_DIS
LIN {X -2.5678,Y 59.1807,Z 71,A 86.6353,B 24.8575,C -2.7544,E1 24.9914,E2 357.1588} C_DIS
LIN {X -4.7626,Y 59.0446,Z 71,A 89.039,B 24.857,C -2.759,E1 24.9846,E2 354.7431} C_DIS
LIN {X -7.8334,Y 58.7159,Z 71,A 92.6417,B 24.8559,C -2.7697,E1 24.9746,E2 351.1124} C_DIS
LIN {X -11.1234,Y 58.1826,Z 71,A 94.9068,B 24.8582,C -2.7481,E1 24.9685,E2 348.8964} C_DIS
LIN {X -14.8835,Y 57.3362,Z 71,A 98.6505,B 24.8585,C -2.745,E1 24.9583,E2 345.155} C_DIS
LIN {X -17.3316,Y 56.6443,Z 71,A 101.3148,B 24.8583,C -2.7463,E1 24.9512,E2 342.4832} C_DIS
LIN {X -19.9657,Y 55.7713,Z 71,A 104.2137,B 24.8583,C -2.7471,E1 24.9435,E2 339.5766} C_DIS
LIN {X -23.903,Y 54.1999,Z 71,A 108.1062,B 24.8593,C -2.7374,E1 24.9335,E2 335.6984} C_DIS
LIN {X -27.5648,Y 52.4321,Z 71,A 112.4314,B 24.8591,C -2.7386,E1 24.9227,E2 331.3587} C_DIS
LIN {X -30.3812,Y 50.8528,Z 71,A 115.3313,B 24.8601,C -2.7289,E1 24.9158,E2 328.4733} C_DIS
LIN {X -33.082,Y 49.138,Z 71,A 118.0564,B 24.8614,C -2.7161,E1 24.9094,E2 325.7698} C_DIS
LIN {X -35.52,Y 47.4055,Z 71,A 121.3413,B 24.8614,C -2.7176,E1 24.902,E2 322.4699} C_DIS
LIN {X -38.3779,Y 45.1229,Z 71,A 124.381,B 24.863,C -2.7008,E1 24.8955,E2 319.4588} C_DIS
LIN {X -40.6611,Y 43.0761,Z 71,A 127.7651,B 24.863,C -2.7017,E1 24.8885,E2 316.0589} C_DIS
LIN {X -43.1955,Y 40.5351,Z 71,A 131.425,B 24.8634,C -2.6968,E1 24.8814,E2 312.3949} C_DIS
LIN {X -45.6991,Y 37.6906,Z 71,A 134.7916,B 24.8649,C -2.6821,E1 24.8753,E2 309.048} C_DIS
LIN {X -47.61,Y 35.2465,Z 71,A 137.96,B 24.8654,C -2.6772,E1 24.87,E2 305.8762} C_DIS
LIN {X -49.1543,Y 33.058,Z 71,A 140.2656,B 24.8666,C -2.6651,E1 24.8663,E2 303.5881} C_DIS
LIN {X -50.4807,Y 30.9941,Z 71,A 143.0088,B 24.8666,C -2.6651,E1 24.8623,E2 300.8309} C_DIS
LIN {X -52.413,Y 27.6011,Z 71,A 147.0606,B 24.8672,C -2.6592,E1 24.8568,E2 296.7719} C_DIS
LIN {X -53.9032,Y 24.5653,Z 71,A 150.0617,B 24.8687,C -2.6448,E1 24.8533,E2 293.7889} C_DIS
LIN {X -55.1724,Y 21.5619,Z 71,A 153.3454,B 24.8694,C -2.6376,E1 24.8499,E2 290.504} C_DIS
LIN {X -56.1939,Y 18.7411,Z 71,A 156.191,B 24.8703,C -2.6278,E1 24.8473,E2 287.6657} C_DIS
LIN {X -57.1839,Y 15.4577,Z 71,A 159.3798,B 24.8716,C -2.6153,E1 24.8448,E2 284.4883} C_DIS
LIN {X -58.1636,Y 11.2222,Z 71,A 163.8788,B 24.8724,C -2.6073,E1 24.8422,E2 279.982} C_DIS
LIN {X -58.7711,Y 7.4124,Z 71,A 167.449,B 24.8738,C -2.5927,E1 24.8408,E2 276.4253} C_DIS
LIN {X -59.0794,Y 4.3221,Z 71,A 170.3623,B 24.8749,C -2.5816,E1 24.8401,E2 273.5211} C_DIS
LIN {X -59.1876,Y 2.4072,Z 71,A 172.9478,B 24.8742,C -2.5886,E1 24.8398,E2 270.9032} C_DIS
LIN {X -59.2005,Y -2.0771,Z 71,A 176.9445,B 24.8761,C -2.5689,E1 24.84,E2 266.9296} C_DIS
LIN {X -58.9736,Y -5.5739,Z 71,A -179.9604,B 24.8776,C -2.5531,E1 24.8407,E2 263.8536} C_DIS
LIN {X -58.7323,Y -7.7117,Z 71,A -177.5809,B 24.8777,C -2.552,E1 24.8415,E2 261.4627} C_DIS
LIN {X -58.1157,Y -11.4711,Z 71,A -174.3237,B 24.8795,C -2.5331,E1 24.8431,E2 258.2313} C_DIS
LIN {X -57.6618,Y -13.5688,Z 71,A -172.1404,B 24.88,C -2.5287,E1 24.8445,E2 256.0456} C_DIS
LIN {X -56.9106,Y -16.4383,Z 71,A -169.3731,B 24.881,C -2.5183,E1 24.8465,E2 253.2871} C_DIS
LIN {X -55.8912,Y -19.6243,Z 71,A -165.8783,B 24.8814,C -2.5135,E1 24.8496,E2 249.7839} C_DIS
LIN {X -55.1826,Y -21.5369,Z 71,A -163.6718,B 24.8816,C -2.512,E1 24.8518,E2 247.5685} C_DIS
LIN {X -53.7418,Y -24.9153,Z 71,A -160.4369,B 24.883,C -2.4964,E1 24.8555,E2 244.3532} C_DIS
LIN {X -51.8566,Y -28.6341,Z 71,A -156.3841,B 24.884,C -2.4858,E1 24.8607,E2 240.304} C_DIS
LIN {X -49.9698,Y -31.8121,Z 71,A -151.9371,B 24.8834,C -2.4926,E1 24.8673,E2 235.8181} C_DIS
LIN {X -47.8292,Y -34.9473,Z 71,A -148.9022,B 24.8853,C -2.4719,E1 24.8721,E2 232.8178} C_DIS
LIN {X -45.604,Y -37.805,Z 71,A -145.7105,B 24.8866,C -2.458,E1 24.8777,E2 229.6444} C_DIS
LIN {X -43.1178,Y -40.6177,Z 71,A -141.8359,B 24.8869,C -2.4545,E1 24.8849,E2 225.7608} C_DIS
LIN {X -41.7169,Y -42.0554,Z 71,A -139.7726,B 24.8871,C -2.4527,E1 24.889,E2 223.6929} C_DIS
LIN {X -39.363,Y -44.2664,Z 71,A -136.6026,B 24.8876,C -2.4475,E1 24.8955,E2 220.5227} C_DIS
LIN {X -37.1633,Y -46.1287,Z 71,A -133.3066,B 24.8871,C -2.4521,E1 24.9027,E2 217.2032} C_DIS
LIN {X -33.6055,Y -48.7813,Z 71,A -129.3816,B 24.8885,C -2.4379,E1 24.9116,E2 213.2985} C_DIS
LIN {X -30.8045,Y -50.5967,Z 71,A -126.2777,B 24.8891,C -2.4307,E1 24.9189,E2 210.2019} C_DIS
LIN {X -28.1852,Y -52.1013,Z 71,A -123.4713,B 24.8897,C -2.4246,E1 24.9258,E2 207.4021} C_DIS
LIN {X -25.1788,Y -53.6191,Z 71,A -120.2722,B 24.8901,C -2.4195,E1 24.9338,E2 204.2066} C_DIS
LIN {X -22.3796,Y -54.8461,Z 71,A -117.3014,B 24.8904,C -2.4168,E1 24.9414,E2 201.2355} C_DIS
LIN {X -19.9717,Y -55.7691,Z 71,A -114.3247,B 24.8897,C -2.4243,E1 24.9493,E2 198.235} C_DIS
LIN {X -17.4704,Y -56.6015,Z 71,A -111.5922,B 24.8895,C -2.4262,E1 24.9566,E2 195.4932} C_DIS
LIN {X -12.1627,Y -57.9748,Z 71,A -106.2472,B 24.8897,C -2.4244,E1 24.9711,E2 190.1454} C_DIS
LIN {X -5.6687,Y -58.9649,Z 71,A -100.7368,B 24.8914,C -2.4055,E1 24.9863,E2 184.6756} C_DIS
LIN {X -2.5537,Y -59.1813,Z 71,A -97.0076,B 24.89,C -2.4206,E1 24.9968,E2 180.9094} C_DIS
LIN {X 0.3248,Y -59.2353,Z 71,A -95.3701,B 24.8922,C -2.3969,E1 25.0012,E2 179.3282} C_DIS
Enddeposition()
LIN {X 0.3248,Y -59.2353,Z 71,A -95.3701,B 24.8922,C -2.3969,E1 25.0012,E2 179.3282} C_DIS
Startdeposition()
$VEL.CP = VEL_PRINT
LIN {X -0.3016,Y -58.3167,Z 71,A -96.9503,B 24.8925,C -2.3931,E1 24.9967,E2 180.9175} C_DIS
LIN {X -3.9472,Y -58.1837,Z 71,A -100.1011,B 24.8918,C -2.4016,E1 24.988,E2 184.0491} C_DIS
LIN {X -7.6066,Y -57.8193,Z 71,A -103.6055,B 24.8915,C -2.4041,E1 24.9783,E2 187.5494} C_DIS
LIN {X -10.0356,Y -57.4482,Z 71,A -106.7608,B 24.8928,C -2.3902,E1 24.9695,E2 190.7408} C_DIS
LIN {X -14.302,Y -56.5369,Z 71,A -110.1253,B 24.891,C -2.4103,E1 24.9605,E2 194.0619} C_DIS
LIN {X -16.7828,Y -55.8507,Z 71,A -113.3608,B 24.8921,C -2.3982,E1 24.9517,E2 197.3314} C_DIS
LIN {X -19.6992,Y -54.8904,Z 71,A -116.1892,B 24.8915,C -2.4043,E1 24.9442,E2 200.1508} C_DIS
LIN {X -22.6246,Y -53.7499,Z 71,A -119.0738,B 24.8909,C -2.4111,E1 24.9368,E2 203.0255} C_DIS
LIN {X -24.4941,Y -52.9243,Z 71,A -122.3432,B 24.8928,C -2.3897,E1 24.9284,E2 206.354} C_DIS
LIN {X -27.8474,Y -51.2391,Z 71,A -124.6245,B 24.89,C -2.4205,E1 24.9229,E2 208.5682} C_DIS
LIN {X -29.4376,Y -50.3431,Z 71,A -126.6833,B 24.8903,C -2.418,E1 24.9179,E2 210.639} C_DIS
LIN {X -31.8174,Y -48.8742,Z 71,A -130.1756,B 24.8911,C -2.4085,E1 24.9096,E2 214.1653} C_DIS
LIN {X -35.5662,Y -46.2166,Z 71,A -134.1674,B 24.8896,C -2.4257,E1 24.9007,E2 218.1303} C_DIS
LIN {X -37.7328,Y -44.4654,Z 71,A -137.4269,B 24.89,C -2.4214,E1 24.8937,E2 221.4126} C_DIS
LIN {X -40.7306,Y -41.738,Z 71,A -140.6734,B 24.888,C -2.4424,E1 24.8872,E2 224.6221} C_DIS
LIN {X -42.4569,Y -39.9792,Z 71,A -143.5615,B 24.8883,C -2.4393,E1 24.8815,E2 227.5302} C_DIS
LIN {X -44.4535,Y -37.7468,Z 71,A -145.8619,B 24.8867,C -2.4573,E1 24.8774,E2 229.7981} C_DIS
LIN {X -45.9312,Y -35.9344,Z 71,A -148.6702,B 24.887,C -2.4536,E1 24.8724,E2 232.6283} C_DIS
LIN {X -47.6201,Y -33.6647,Z 71,A -151.8882,B 24.887,C -2.4527,E1 24.8672,E2 235.8642} C_DIS
LIN {X -50.1089,Y -29.8339,Z 71,A -155.4301,B 24.8845,C -2.4806,E1 24.862,E2 239.3575} C_DIS
LIN {X -51.1431,Y -28.0245,Z 71,A -158.1515,B 24.8851,C -2.4744,E1 24.8583,E2 242.1081} C_DIS
LIN {X -52.7215,Y -24.9282,Z 71,A -161.0845,B 24.8834,C -2.492,E1 24.8547,E2 245.0148} C_DIS
LIN {X -53.5214,Y -23.1603,Z 71,A -163.7366,B 24.8841,C -2.4846,E1 24.8517,E2 247.6991} C_DIS
LIN {X -54.8196,Y -19.8932,Z 71,A -166.8149,B 24.8826,C -2.5009,E1 24.8487,E2 250.7558} C_DIS
LIN {X -55.8126,Y -16.9115,Z 71,A -170.0762,B 24.882,C -2.5071,E1 24.8459,E2 254.0212} C_DIS
LIN {X -56.8925,Y -12.8142,Z 71,A -174.0334,B 24.8805,C -2.5231,E1 24.8433,E2 257.9632} C_DIS
LIN {X -57.6843,Y -8.5733,Z 71,A -177.9637,B 24.8788,C -2.5412,E1 24.8414,E2 261.8735} C_DIS
LIN {X -57.9463,Y -6.5724,Z 71,A 179.7825,B 24.8786,C -2.5428,E1 24.8406,E2 264.1368} C_DIS
LIN {X -58.1948,Y -3.7836,Z 71,A 176.9683,B 24.8779,C -2.5504,E1 24.84,E2 266.9499} C_DIS
LIN {X -58.3194,Y -0.0686,Z 71,A 172.801,B 24.8776,C -2.5533,E1 24.8398,E2 271.1354} C_DIS
LIN {X -58.1957,Y 3.7696,Z 71,A 169.4656,B 24.8758,C -2.5725,E1 24.8403,E2 274.4449} C_DIS
LIN {X -57.9397,Y 6.6284,Z 71,A 166.2441,B 24.8755,C -2.5748,E1 24.8412,E2 277.6804} C_DIS
LIN {X -57.2686,Y 11.0105,Z 71,A 161.882,B 24.8742,C -2.5883,E1 24.8433,E2 282.0358} C_DIS
LIN {X -56.5454,Y 14.2691,Z 71,A 159.1193,B 24.8724,C -2.6071,E1 24.845,E2 284.7699} C_DIS
LIN {X -55.386,Y 18.2599,Z 71,A 155.2164,B 24.8708,C -2.6227,E1 24.8481,E2 288.658} C_DIS
LIN {X -53.9805,Y 22.0689,Z 71,A 150.687,B 24.8706,C -2.6257,E1 24.8527,E2 293.2058} C_DIS
LIN {X -52.4406,Y 25.5144,Z 71,A 147.5069,B 24.8686,C -2.6455,E1 24.8563,E2 296.3559} C_DIS
LIN {X -50.7268,Y 28.7718,Z 71,A 142.9979,B 24.8691,C -2.6408,E1 24.8624,E2 300.9} C_DIS
LIN {X -48.4886,Y 32.4023,Z 71,A 139.3655,B 24.867,C -2.6618,E1 24.8678,E2 304.5005} C_DIS
LIN {X -46.8552,Y 34.7196,Z 71,A 136.1297,B 24.867,C -2.6616,E1 24.8731,E2 307.7525} C_DIS
LIN {X -44.8956,Y 37.2198,Z 71,A 132.7054,B 24.8667,C -2.6645,E1 24.8792,E2 311.186} C_DIS
LIN {X -42.2161,Y 40.2347,Z 71,A 129.3512,B 24.8647,C -2.6846,E1 24.8854,E2 314.5068} C_DIS
LIN {X -40.3603,Y 42.095,Z 71,A 126.6939,B 24.8642,C -2.6894,E1 24.8907,E2 317.1639} C_DIS
LIN {X -38.6774,Y 43.6471,Z 71,A 124.4487,B 24.8637,C -2.6945,E1 24.8954,E2 319.4059} C_DIS
LIN {X -35.22,Y 46.4804,Z 71,A 120.2412,B 24.8624,C -2.7071,E1 24.9045,E2 323.599} C_DIS
LIN {X -33.4322,Y 47.7833,Z 71,A 117.8428,B 24.8624,C -2.7074,E1 24.91,E2 326.0049} C_DIS
LIN {X -30.0272,Y 49.9939,Z 71,A 113.9318,B 24.8614,C -2.7162,E1 24.9192,E2 329.9074} C_DIS
LIN {X -25.7965,Y 52.3018,Z 71,A 108.9061,B 24.8612,C -2.7187,E1 24.9316,E2 334.941} C_DIS
LIN {X -22.2198,Y 53.9191,Z 71,A 104.874,B 24.8609,C -2.721,E1 24.942,E2 338.9771} C_DIS
LIN {X -18.8123,Y 55.2001,Z 71,A 101.1581,B 24.8608,C -2.7229,E1 24.9518,E2 342.6959} C_DIS
LIN {X -14.3741,Y 56.5184,Z 71,A 97.3691,B 24.8588,C -2.7418,E1 24.9618,E2 346.4458} C_DIS
LIN {X -12.2045,Y 57.0265,Z 71,A 94.9344,B 24.8591,C -2.7391,E1 24.9685,E2 348.8901} C_DIS
LIN {X -8.8627,Y 57.6401,Z 71,A 91.1279,B 24.8598,C -2.7326,E1 24.979,E2 352.7157} C_DIS
LIN {X -5.1173,Y 58.093,Z 71,A 87.8341,B 24.8587,C -2.7425,E1 24.9881,E2 355.988} C_DIS
LIN {X -2.2869,Y 58.273,Z 71,A 84.3962,B 24.8599,C -2.7308,E1 24.9978,E2 359.4544} C_DIS
LIN {X 2.2384,Y 58.2751,Z 71,A 80.5092,B 24.8588,C -2.7423,E1 25.0085,E2 363.3134} C_DIS
LIN {X 4.9056,Y 58.1113,Z 71,A 77.9732,B 24.8586,C -2.744,E1 25.0156,E2 365.8443} C_DIS
LIN {X 7.705,Y 57.8066,Z 71,A 74.9398,B 24.8592,C -2.7382,E1 25.024,E2 368.8892} C_DIS
LIN {X 11.6507,Y 57.1419,Z 71,A 70.8764,B 24.8596,C -2.734,E1 25.0352,E2 372.9579} C_DIS
LIN {X 15.5668,Y 56.2017,Z 71,A 67.4072,B 24.8588,C -2.7416,E1 25.0445,E2 376.4038} C_DIS
LIN {X 18.1215,Y 55.4307,Z 71,A 64.6472,B 24.8593,C -2.7367,E1 25.0519,E2 379.1702} C_DIS
LIN {X 20.7942,Y 54.4844,Z 71,A 62.1538,B 24.859,C -2.7403,E1 25.0584,E2 381.6499} C_DIS
LIN {X 23.6053,Y 53.3259,Z 71,A 58.9347,B 24.8598,C -2.7323,E1 25.0667,E2 384.8804} C_DIS
LIN {X 25.8949,Y 52.253,Z 71,A 56.5756,B 24.8598,C -2.732,E1 25.0726,E2 387.2341} C_DIS
LIN {X 27.718,Y 51.3093,Z 71,A 54.4465,B 24.8603,C -2.727,E1 25.0779,E2 389.369} C_DIS
LIN {X 30.8092,Y 49.5149,Z 71,A 51.0241,B 24.8607,C -2.7238,E1 25.0861,E2 392.7884} C_DIS
LIN {X 34.189,Y 47.2448,Z 71,A 47.1963,B 24.8609,C -2.721,E1 25.0949,E2 396.6098} C_DIS
LIN {X 36.8397,Y 45.2082,Z 71,A 44.0074,B 24.8613,C -2.7173,E1 25.1019,E2 399.7958} C_DIS
LIN {X 38.2643,Y 44.0089,Z 71,A 41.8524,B 24.8624,C -2.7067,E1 25.1065,E2 401.9675} C_DIS
LIN {X 40.3794,Y 42.0766,Z 71,A 38.2608,B 24.8647,C -2.684,E1 25.1139,E2 405.598} C_DIS
LIN {X 43.0784,Y 39.3091,Z 71,A 35.5226,B 24.8632,C -2.6991,E1 25.119,E2 408.2885} C_DIS
LIN {X 45.4207,Y 36.5776,Z 71,A 31.8188,B 24.8644,C -2.6873,E1 25.1257,E2 412.0034} C_DIS
LIN {X 47.0336,Y 34.4784,Z 71,A 29.3539,B 24.8647,C -2.6841,E1 25.1298,E2 414.464} C_DIS
LIN {X 48.5403,Y 32.3215,Z 71,A 26.3426,B 24.8663,C -2.6681,E1 25.1346,E2 417.4983} C_DIS
LIN {X 50.7403,Y 28.7465,Z 71,A 22.54,B 24.8667,C -2.6646,E1 25.14,E2 421.2897} C_DIS
LIN {X 51.8414,Y 26.7101,Z 71,A 20.4641,B 24.8668,C -2.663,E1 25.1427,E2 423.3585} C_DIS
LIN {X 52.961,Y 24.4152,Z 71,A 18.0859,B 24.8672,C -2.659,E1 25.1456,E2 425.7332} C_DIS
LIN {X 53.9542,Y 22.1334,Z 71,A 15.1132,B 24.8691,C -2.6401,E1 25.1488,E2 428.7346} C_DIS
LIN {X 55.2272,Y 18.732,Z 71,A 11.7688,B 24.8696,C -2.6348,E1 25.152,E2 432.0726} C_DIS
LIN {X 56.0887,Y 15.9684,Z 71,A 8.3176,B 24.8719,C -2.6125,E1 25.1547,E2 435.5568} C_DIS
LIN {X 56.8872,Y 12.8397,Z 71,A 5.3106,B 24.8724,C -2.6066,E1 25.1566,E2 438.5602} C_DIS
LIN {X 57.7496,Y 8.1186,Z 71,A 1.1555,B 24.8726,C -2.605,E1 25.1585,E2 442.6947} C_DIS
LIN {X 58.1296,Y 4.6765,Z 71,A -2.5333,B 24.8743,C -2.5878,E1 25.1595,E2 446.4024} C_DIS
LIN {X 58.3074,Y 1.0777,Z 71,A -6.2188,B 24.8757,C -2.5733,E1 25.1598,E2 450.1002} C_DIS
LIN {X 58.276,Y -2.217,Z 71,A -9.4378,B 24.8766,C -2.5634,E1 25.1595,E2 453.3233} C_DIS
LIN {X 57.9753,Y -6.3123,Z 71,A -12.8348,B 24.8764,C -2.5655,E1 25.1587,E2 456.6954} C_DIS
LIN {X 57.6378,Y -8.8774,Z 71,A -15.5401,B 24.8776,C -2.5537,E1 25.1576,E2 459.4128} C_DIS
LIN {X 57.1474,Y -11.6235,Z 71,A -18.194,B 24.8782,C -2.5471,E1 25.1562,E2 462.0667} C_DIS
LIN {X 56.4757,Y -14.5403,Z 71,A -20.6973,B 24.8782,C -2.5481,E1 25.1546,E2 464.5531} C_DIS
LIN {X 55.9127,Y -16.5738,Z 71,A -23.1881,B 24.8797,C -2.5319,E1 25.1527,E2 467.0679} C_DIS
LIN {X 55.0873,Y -19.1401,Z 71,A -25.7399,B 24.8802,C -2.5261,E1 25.1504,E2 469.6191} C_DIS
LIN {X 53.9262,Y -22.2022,Z 71,A -29.3891,B 24.8821,C -2.5064,E1 25.1467,E2 473.2946} C_DIS
LIN {X 52.5254,Y -25.338,Z 71,A -32.4961,B 24.8824,C -2.5025,E1 25.143,E2 476.3939} C_DIS
LIN {X 50.9255,Y -28.4168,Z 71,A -35.5568,B 24.8826,C -2.5007,E1 25.139,E2 479.4427} C_DIS
LIN {X 49.667,Y -30.565,Z 71,A -38.8704,B 24.8851,C -2.474,E1 25.1341,E2 482.8028} C_DIS
LIN {X 47.2303,Y -34.2099,Z 71,A -43.0465,B 24.8859,C -2.4653,E1 25.1274,E2 486.979} C_DIS
LIN {X 44.2662,Y -37.9666,Z 71,A -47.1395,B 24.8858,C -2.4669,E1 25.1202,E2 491.0492} C_DIS
LIN {X 41.8459,Y -40.6188,Z 71,A -51.0346,B 24.8873,C -2.45,E1 25.1127,E2 494.9675} C_DIS
LIN {X 39.6853,Y -42.7328,Z 71,A -53.8422,B 24.8877,C -2.4466,E1 25.1071,E2 497.7713} C_DIS
LIN {X 36.8836,Y -45.1726,Z 71,A -57.1493,B 24.8877,C -2.4462,E1 25.1,E2 501.0665} C_DIS
LIN {X 34.1084,Y -47.3036,Z 71,A -61.1485,B 24.8895,C -2.4267,E1 25.091,E2 505.0977} C_DIS
LIN {X 31.5912,Y -49.0197,Z 71,A -64.3839,B 24.8905,C -2.4157,E1 25.0834,E2 508.3486} C_DIS
LIN {X 27.7946,Y -51.2677,Z 71,A -68.1113,B 24.89,C -2.4213,E1 25.0744,E2 512.0516} C_DIS
LIN {X 25.1388,Y -52.6204,Z 71,A -70.7614,B 24.8899,C -2.4227,E1 25.0678,E2 514.6914} C_DIS
LIN {X 22.8176,Y -53.6686,Z 71,A -73.1281,B 24.8899,C -2.4219,E1 25.0618,E2 517.0542} C_DIS
LIN {X 19.7816,Y -54.8603,Z 71,A -76.9575,B 24.8915,C -2.4042,E1 25.0517,E2 520.9172} C_DIS
LIN {X 16.7191,Y -55.8696,Z 71,A -79.5622,B 24.8908,C -2.4125,E1 25.0448,E2 523.4975} C_DIS
LIN {X 13.1248,Y -56.8213,Z 71,A -83.3732,B 24.8914,C -2.4055,E1 25.0345,E2 527.3193} C_DIS
LIN {X 10.9971,Y -57.2712,Z 71,A -85.5283,B 24.8916,C -2.4033,E1 25.0285,E2 529.477} C_DIS
LIN {X 8.2382,Y -57.7326,Z 71,A -88.8006,B 24.8928,C -2.3905,E1 25.0194,E2 532.7767} C_DIS
LIN {X 3.8306,Y -58.1916,Z 71,A -92.7447,B 24.8922,C -2.3968,E1 25.0085,E2 536.7038} C_DIS
LIN {X 1.1758,Y -58.3057,Z 71,A -95.2548,B 24.8921,C -2.398,E1 25.0015,E2 539.2104} C_DIS
LIN {X 1.1758,Y -58.3057,Z 71,A -95.2548,B 24.8921,C -2.398,E1 25.0015,E2 539.2104} C_DIS
Enddeposition()
LIN {X 0.3166,Y -57.3948,Z 71,A -95.6629,B 24.8898,C -2.4227,E1 25.0005,E2 539.5596} C_DIS
Startdeposition()
$VEL.CP = VEL_PRINT
LIN {X 2.2196,Y -57.3561,Z 71,A -92.9167,B 24.8882,C -2.4405,E1 25.0083,E2 536.7717} C_DIS
LIN {X 6.2795,Y -57.0543,Z 71,A -88.5376,B 24.8874,C -2.4491,E1 25.0205,E2 532.3746} C_DIS
LIN {X 9.4608,Y -56.6135,Z 71,A -85.686,B 24.8879,C -2.444,E1 25.0284,E2 529.538} C_DIS
LIN {X 12.0425,Y -56.1214,Z 71,A -83.0629,B 24.8877,C -2.4462,E1 25.0356,E2 526.9129} C_DIS
LIN {X 14.4208,Y -55.5573,Z 71,A -80.5139,B 24.8873,C -2.4509,E1 25.0425,E2 524.3565} C_DIS
LIN {X 17.008,Y -54.8208,Z 71,A -77.3593,B 24.886,C -2.4641,E1 25.051,E2 521.1762} C_DIS
LIN {X 21.8766,Y -53.0667,Z 71,A -73.0746,B 24.8872,C -2.4518,E1 25.0621,E2 516.9298} C_DIS
LIN {X 24.6128,Y -51.8544,Z 71,A -69.157,B 24.8849,C -2.4767,E1 25.0721,E2 512.9631} C_DIS
LIN {X 28.2456,Y -49.9687,Z 71,A -65.6489,B 24.8854,C -2.4709,E1 25.0807,E2 509.4789} C_DIS
LIN {X 30.0135,Y -48.9269,Z 71,A -63.6718,B 24.8852,C -2.4731,E1 25.0854,E2 507.5028} C_DIS
LIN {X 31.9154,Y -47.7086,Z 71,A -61.0239,B 24.884,C -2.4862,E1 25.0916,E2 504.8326} C_DIS
LIN {X 35.8517,Y -44.8259,Z 71,A -56.8885,B 24.8846,C -2.4798,E1 25.1008,E2 500.7272} C_DIS
LIN {X 37.8581,Y -43.1437,Z 71,A -53.4813,B 24.8823,C -2.5036,E1 25.1081,E2 497.2771} C_DIS
LIN {X 41.437,Y -39.719,Z 71,A -48.424,B 24.881,C -2.518,E1 25.1181,E2 492.2072} C_DIS
LIN {X 43.5892,Y -37.3444,Z 71,A -45.2537,B 24.8803,C -2.5254,E1 25.1239,E2 489.0336} C_DIS
LIN {X 46.6212,Y -33.4826,Z 71,A -40.9673,B 24.8803,C -2.5242,E1 25.1311,E2 484.7704} C_DIS
LIN {X 48.5068,Y -30.6887,Z 71,A -37.6605,B 24.8796,C -2.5321,E1 25.1361,E2 481.4614} C_DIS
LIN {X 49.8835,Y -28.3951,Z 71,A -35.3168,B 24.8796,C -2.5321,E1 25.1394,E2 479.1296} C_DIS
LIN {X 51.3722,Y -25.6027,Z 71,A -31.8698,B 24.8781,C -2.548,E1 25.1439,E2 475.6634} C_DIS
LIN {X 53.0374,Y -21.9467,Z 71,A -27.3457,B 24.8758,C -2.572,E1 25.149,E2 471.1074} C_DIS
LIN {X 54.1978,Y -18.8998,Z 71,A -24.886,B 24.8767,C -2.5633,E1 25.1513,E2 468.682} C_DIS
LIN {X 55.1803,Y -15.8038,Z 71,A -21.6609,B 24.8757,C -2.5729,E1 25.154,E2 465.4526} C_DIS
LIN {X 55.7729,Y -13.5637,Z 71,A -19.1485,B 24.8746,C -2.5847,E1 25.1557,E2 462.9266} C_DIS
LIN {X 56.3603,Y -10.8681,Z 71,A -16.3205,B 24.8736,C -2.5951,E1 25.1573,E2 460.0906} C_DIS
LIN {X 56.8421,Y -7.9734,Z 71,A -13.9402,B 24.8739,C -2.5915,E1 25.1583,E2 457.7327} C_DIS
LIN {X 57.0816,Y -6.0243,Z 71,A -10.8725,B 24.8708,C -2.6237,E1 25.1593,E2 454.6073} C_DIS
LIN {X 57.3702,Y -1.8042,Z 71,A -7.2715,B 24.8708,C -2.6224,E1 25.1598,E2 451.0306} C_DIS
LIN {X 57.3971,Y 0.5178,Z 71,A -5.0735,B 24.8704,C -2.6269,E1 25.1598,E2 448.8351} C_DIS
LIN {X 57.3098,Y 3.1912,Z 71,A -2.2875,B 24.8693,C -2.638,E1 25.1594,E2 446.0394} C_DIS
LIN {X 56.991,Y 6.8297,Z 71,A 1.2693,B 24.8684,C -2.6473,E1 25.1584,E2 442.4817} C_DIS
LIN {X 56.435,Y 10.4778,Z 71,A 5.3316,B 24.8664,C -2.6674,E1 25.1565,E2 438.3955} C_DIS
LIN {X 55.8308,Y 13.3264,Z 71,A 8.1468,B 24.8657,C -2.6741,E1 25.1547,E2 435.5809} C_DIS
LIN {X 54.9865,Y 16.465,Z 71,A 11.0555,B 24.8655,C -2.676,E1 25.1525,E2 432.6845} C_DIS
LIN {X 54.1198,Y 19.1222,Z 71,A 13.8003,B 24.8648,C -2.6831,E1 25.15,E2 429.9384} C_DIS
LIN {X 53.0804,Y 21.8429,Z 71,A 16.7122,B 24.864,C -2.6915,E1 25.147,E2 427.0227} C_DIS
LIN {X 52.2105,Y 23.8482,Z 71,A 18.7424,B 24.8637,C -2.6941,E1 25.1447,E2 424.9974} C_DIS
LIN {X 50.6978,Y 26.914,Z 71,A 22.3951,B 24.8622,C -2.7089,E1 25.1401,E2 421.3291} C_DIS
LIN {X 49.1473,Y 29.6508,Z 71,A 25.391,B 24.8617,C -2.7138,E1 25.1358,E2 418.3369} C_DIS
LIN {X 47.9055,Y 31.6173,Z 71,A 27.7348,B 24.861,C -2.7202,E1 25.1323,E2 415.9898} C_DIS
LIN {X 45.2267,Y 35.3443,Z 71,A 31.8921,B 24.8609,C -2.7217,E1 25.1254,E2 411.8489} C_DIS
LIN {X 43.8529,Y 37.0348,Z 71,A 34.7674,B 24.8587,C -2.7424,E1 25.1202,E2 408.9378} C_DIS
LIN {X 41.2822,Y 39.8795,Z 71,A 38.6313,B 24.8578,C -2.7515,E1 25.1128,E2 405.0693} C_DIS
LIN {X 38.5811,Y 42.4992,Z 71,A 42.0004,B 24.8579,C -2.7504,E1 25.106,E2 401.7164} C_DIS
LIN {X 36.443,Y 44.3464,Z 71,A 44.9376,B 24.8571,C -2.7583,E1 25.0997,E2 398.7719} C_DIS
LIN {X 33.9721,Y 46.2655,Z 71,A 48.0415,B 24.8566,C -2.7633,E1 25.0928,E2 395.6673} C_DIS
LIN {X 30.9779,Y 48.3215,Z 71,A 51.9317,B 24.8554,C -2.7747,E1 25.0837,E2 391.7629} C_DIS
LIN {X 27.7085,Y 50.2686,Z 71,A 55.321,B 24.8558,C -2.7712,E1 25.0755,E2 388.3921} C_DIS
LIN {X 25.3021,Y 51.5213,Z 71,A 57.8827,B 24.8558,C -2.7715,E1 25.0691,E2 385.8368} C_DIS
LIN {X 21.011,Y 53.4147,Z 71,A 62.5705,B 24.8552,C -2.7766,E1 25.0571,E2 381.1481} C_DIS
LIN {X 18.0481,Y 54.4872,Z 71,A 65.8693,B 24.8546,C -2.7824,E1 25.0484,E2 377.842} C_DIS
LIN {X 15.1439,Y 55.3643,Z 71,A 69.1025,B 24.8539,C -2.7887,E1 25.0397,E2 374.5992} C_DIS
LIN {X 11.1639,Y 56.3033,Z 71,A 73.5049,B 24.853,C -2.7972,E1 25.0276,E2 370.1823} C_DIS
LIN {X 7.2772,Y 56.9354,Z 71,A 76.8216,B 24.8542,C -2.7857,E1 25.0185,E2 366.8959} C_DIS
LIN {X 4.4579,Y 57.2253,Z 71,A 79.6094,B 24.8542,C -2.7851,E1 25.0108,E2 364.1111} C_DIS
LIN {X 2.1269,Y 57.3601,Z 71,A 82.426,B 24.8533,C -2.7947,E1 25.0029,E2 361.2726} C_DIS
LIN {X -2.0993,Y 57.3611,Z 71,A 86.2677,B 24.8542,C -2.7862,E1 24.9922,E2 357.4509} C_DIS
LIN {X -5.0451,Y 57.1769,Z 71,A 89.1831,B 24.8544,C -2.7843,E1 24.9841,E2 354.5388} C_DIS
LIN {X -7.3464,Y 56.9265,Z 71,A 92.4311,B 24.8526,C -2.8012,E1 24.975,E2 351.2482} C_DIS
LIN {X -10.748,Y 56.3834,Z 71,A 94.8928,B 24.8549,C -2.7797,E1 24.9683,E2 348.835} C_DIS
LIN {X -12.606,Y 55.9981,Z 71,A 96.7603,B 24.8551,C -2.7775,E1 24.9633,E2 346.9704} C_DIS
LIN {X -15.6328,Y 55.2287,Z 71,A 100.3385,B 24.8545,C -2.7831,E1 24.9536,E2 343.3733} C_DIS
LIN {X -19.1693,Y 54.1032,Z 71,A 103.6619,B 24.8557,C -2.7715,E1 24.9448,E2 340.0714} C_DIS
LIN {X -23.3274,Y 52.4452,Z 71,A 108.7934,B 24.8551,C -2.7776,E1 24.9315,E2 334.9136} C_DIS
LIN {X -26.1807,Y 51.08,Z 71,A 111.8027,B 24.8559,C -2.7698,E1 24.9241,E2 331.9148} C_DIS
LIN {X -29.6727,Y 49.134,Z 71,A 116.2365,B 24.8558,C -2.7708,E1 24.9134,E2 327.4651} C_DIS
LIN {X -32.512,Y 47.3038,Z 71,A 118.5132,B 24.8585,C -2.7445,E1 24.9082,E2 325.2436} C_DIS
LIN {X -35.0032,Y 45.4903,Z 71,A 122.2984,B 24.8579,C -2.7509,E1 24.8997,E2 321.4296} C_DIS
LIN {X -38.046,Y 42.9791,Z 71,A 125.4746,B 24.8602,C -2.7288,E1 24.8931,E2 318.294} C_DIS
LIN {X -39.5388,Y 41.6095,Z 71,A 127.829,B 24.86,C -2.73,E1 24.8882,E2 315.9271} C_DIS
LIN {X -41.6627,Y 39.4816,Z 71,A 130.9374,B 24.8606,C -2.7247,E1 24.8822,E2 312.818} C_DIS
LIN {X -44.2965,Y 36.503,Z 71,A 134.8137,B 24.8618,C -2.713,E1 24.8752,E2 308.9519} C_DIS
LIN {X -47.231,Y 32.6168,Z 71,A 140.2551,B 24.8621,C -2.7101,E1 24.8662,E2 303.491} C_DIS
LIN {X -50.043,Y 28.1125,Z 71,A 145.4764,B 24.8637,C -2.6938,E1 24.8588,E2 298.2818} C_DIS
LIN {X -51.4047,Y 25.5374,Z 71,A 148.6896,B 24.8641,C -2.6906,E1 24.8548,E2 295.0589} C_DIS
LIN {X -53.2582,Y 21.406,Z 71,A 152.5163,B 24.8666,C -2.6653,E1 24.8506,E2 291.2716} C_DIS
LIN {X -54.2538,Y 18.7402,Z 71,A 155.3324,B 24.8675,C -2.6563,E1 24.848,E2 288.4611} C_DIS
LIN {X -55.111,Y 16.0454,Z 71,A 158.0278,B 24.8686,C -2.6454,E1 24.8458,E2 285.776} C_DIS
LIN {X -56.0526,Y 12.3568,Z 71,A 162.1717,B 24.8692,C -2.6394,E1 24.843,E2 281.6224} C_DIS
LIN {X -56.8788,Y 7.7144,Z 71,A 166.7201,B 24.8709,C -2.6219,E1 24.841,E2 277.0887} C_DIS
LIN {X -57.1747,Y 5.0687,Z 71,A 169.4458,B 24.8716,C -2.6147,E1 24.8402,E2 274.364} C_DIS
LIN {X -57.3499,Y 2.3643,Z 71,A 171.7123,B 24.8732,C -2.5988,E1 24.8399,E2 272.1218} C_DIS
LIN {X -57.3981,Y 0.4052,Z 71,A 174.4688,B 24.8725,C -2.606,E1 24.8398,E2 269.3314} C_DIS
LIN {X -57.3179,Y -3.0445,Z 71,A 177.5486,B 24.8741,C -2.5891,E1 24.8401,E2 266.2735} C_DIS
LIN {X -57.1165,Y -5.6902,Z 71,A -179.7698,B 24.8749,C -2.5814,E1 24.8408,E2 263.5943} C_DIS
LIN {X -56.7914,Y -8.3306,Z 71,A -177.1546,B 24.8758,C -2.5725,E1 24.8417,E2 260.9848} C_DIS
LIN {X -56.3101,Y -11.1285,Z 71,A -174.397,B 24.8767,C -2.5625,E1 24.8431,E2 258.2347} C_DIS
LIN {X -55.7462,Y -13.6732,Z 71,A -171.4903,B 24.877,C -2.5598,E1 24.845,E2 255.3173} C_DIS
LIN {X -55.0701,Y -16.1832,Z 71,A -168.7948,B 24.8776,C -2.5538,E1 24.847,E2 252.6206} C_DIS
LIN {X -53.7782,Y -20.0643,Z 71,A -165.2594,B 24.8796,C -2.5326,E1 24.8502,E2 249.1158} C_DIS
LIN {X -52.6169,Y -22.9359,Z 71,A -161.26,B 24.8789,C -2.5395,E1 24.8546,E2 245.0778} C_DIS
LIN {X -51.1752,Y -25.9935,Z 71,A -158.329,B 24.8806,C -2.5225,E1 24.8582,E2 242.1714} C_DIS
LIN {X -49.8036,Y -28.5341,Z 71,A -155.5282,B 24.8814,C -2.5135,E1 24.862,E2 239.3775} C_DIS
LIN {X -48.2742,Y -31.0515,Z 71,A -151.922,B 24.881,C -2.5177,E1 24.8674,E2 235.7429} C_DIS
LIN {X -45.9683,Y -34.3734,Z 71,A -148.6829,B 24.8833,C -2.4937,E1 24.8726,E2 232.5452} C_DIS
LIN {X -44.3142,Y -36.4817,Z 71,A -145.306,B 24.8827,C -2.5,E1 24.8786,E2 229.1376} C_DIS
LIN {X -41.618,Y -39.53,Z 71,A -141.6656,B 24.8842,C -2.4836,E1 24.8854,E2 225.5204} C_DIS
LIN {X -39.738,Y -41.4186,Z 71,A -139.2869,B 24.8852,C -2.4731,E1 24.8901,E2 223.1568} C_DIS
LIN {X -36.8476,Y -44.0101,Z 71,A -135.1988,B 24.8855,C -2.4695,E1 24.8987,E2 219.0611} C_DIS
LIN {X -34.5369,Y -45.8454,Z 71,A -132.05,B 24.8857,C -2.468,E1 24.9056,E2 215.9041} C_DIS
LIN {X -31.6022,Y -47.9155,Z 71,A -128.5297,B 24.8863,C -2.4611,E1 24.9137,E2 212.3885} C_DIS
LIN {X -29.1952,Y -49.419,Z 71,A -125.6746,B 24.8867,C -2.4574,E1 24.9205,E2 209.5334} C_DIS
LIN {X -26.7524,Y -50.7829,Z 71,A -123.1618,B 24.8875,C -2.4485,E1 24.9267,E2 207.0347} C_DIS
LIN {X -23.8084,Y -52.2285,Z 71,A -119.7648,B 24.8876,C -2.447,E1 24.9352,E2 203.6326} C_DIS
LIN {X -21.0119,Y -53.4144,Z 71,A -116.4511,B 24.8874,C -2.4494,E1 24.9438,E2 200.3057} C_DIS
LIN {X -18.0821,Y -54.4756,Z 71,A -113.1106,B 24.8872,C -2.4514,E1 24.9527,E2 196.9542} C_DIS
LIN {X -14.4084,Y -55.5608,Z 71,A -110.1759,B 24.889,C -2.4316,E1 24.9605,E2 194.0619} C_DIS
LIN {X -11.1151,Y -56.3127,Z 71,A -106.2875,B 24.8883,C -2.4401,E1 24.9711,E2 190.1483} C_DIS
LIN {X -8.4509,Y -56.7739,Z 71,A -103.5713,B 24.8883,C -2.4397,E1 24.9786,E2 187.4306} C_DIS
LIN {X -5.77,Y -57.1082,Z 71,A -101.2754,B 24.8891,C -2.4313,E1 24.9849,E2 185.1531} C_DIS
LIN {X -3.0996,Y -57.3148,Z 71,A -97.6601,B 24.8873,C -2.4505,E1 24.9951,E2 181.4909} C_DIS
LIN {X 0.3166,Y -57.3948,Z 71,A -95.662,B 24.8899,C -2.4224,E1 25.0005,E2 179.5596} C_DIS
Enddeposition()
LIN {X 0.3166,Y -57.3948,Z 71,A -95.662,B 24.8899,C -2.4224,E1 25.0005,E2 179.5596} C_DIS
Startdeposition()
$VEL.CP = VEL_PRINT
LIN {X -0.5776,Y -56.4772,Z 71,A -97.1879,B 24.8895,C -2.426,E1 24.9963,E2 181.077} C_DIS
LIN {X -3.9587,Y -56.341,Z 71,A -100.4769,B 24.8893,C -2.4286,E1 24.9871,E2 184.3607} C_DIS
LIN {X -6.8101,Y -56.0681,Z 71,A -103.3012,B 24.8891,C -2.4305,E1 24.9793,E2 187.1822} C_DIS
LIN {X -9.3193,Y -55.7055,Z 71,A -105.8371,B 24.8891,C -2.4318,E1 24.9723,E2 189.7171} C_DIS
LIN {X -11.945,Y -55.2021,Z 71,A -108.8242,B 24.8894,C -2.4277,E1 24.9641,E2 192.7174} C_DIS
LIN {X -14.1815,Y -54.6704,Z 71,A -111.0184,B 24.889,C -2.4316,E1 24.9582,E2 194.9056} C_DIS
LIN {X -17.564,Y -53.6785,Z 71,A -114.6973,B 24.889,C -2.4322,E1 24.9483,E2 198.5893} C_DIS
LIN {X -20.9456,Y -52.4515,Z 71,A -118.7045,B 24.8893,C -2.429,E1 24.9379,E2 202.6126} C_DIS
LIN {X -25.2811,Y -50.5061,Z 71,A -123.0428,B 24.888,C -2.4432,E1 24.9269,E2 206.928} C_DIS
LIN {X -27.55,Y -49.3047,Z 71,A -125.7068,B 24.8878,C -2.4456,E1 24.9204,E2 209.594} C_DIS
LIN {X -29.9721,Y -47.871,Z 71,A -128.582,B 24.8874,C -2.4493,E1 24.9135,E2 212.4691} C_DIS
LIN {X -32.3489,Y -46.2981,Z 71,A -131.6333,B 24.8872,C -2.4511,E1 24.9065,E2 215.5264} C_DIS
LIN {X -34.9564,Y -44.3622,Z 71,A -134.7748,B 24.8865,C -2.4595,E1 24.8995,E2 218.6592} C_DIS
LIN {X -37.1038,Y -42.5824,Z 71,A -137.7763,B 24.8862,C -2.4618,E1 24.8931,E2 221.6668} C_DIS
LIN {X -38.8094,Y -41.0342,Z 71,A -139.9632,B 24.8856,C -2.4691,E1 24.8887,E2 223.8455} C_DIS
LIN {X -40.7214,Y -39.1373,Z 71,A -142.743,B 24.8851,C -2.474,E1 24.8833,E2 226.6254} C_DIS
LIN {X -43.2116,Y -36.3706,Z 71,A -146.4808,B 24.8843,C -2.483,E1 24.8764,E2 230.3585} C_DIS
LIN {X -44.8947,Y -34.2707,Z 71,A -149.2622,B 24.8838,C -2.4885,E1 24.8716,E2 233.1398} C_DIS
LIN {X -46.5074,Y -32.0479,Z 71,A -152.1795,B 24.8833,C -2.4932,E1 24.8669,E2 236.0603} C_DIS
LIN {X -47.7675,Y -30.1377,Z 71,A -154.3084,B 24.8825,C -2.5023,E1 24.8637,E2 238.1782} C_DIS
LIN {X -49.1795,Y -27.7741,Z 71,A -157.0787,B 24.8817,C -2.5099,E1 24.8598,E2 240.9446} C_DIS
LIN {X -50.4658,Y -25.3616,Z 71,A -160.7569,B 24.8824,C -2.5026,E1 24.8551,E2 244.66} C_DIS
LIN {X -52.2916,Y -21.3434,Z 71,A -164.4839,B 24.8801,C -2.5274,E1 24.851,E2 248.3484} C_DIS
LIN {X -53.2798,Y -18.7407,Z 71,A -168.2538,B 24.8808,C -2.5203,E1 24.8474,E2 252.1566} C_DIS
LIN {X -54.2802,Y -15.6098,Z 71,A -170.2279,B 24.8777,C -2.5521,E1 24.8459,E2 254.066} C_DIS
LIN {X -55.3396,Y -11.291,Z 71,A -174.9972,B 24.8768,C -2.5615,E1 24.8428,E2 258.8408} C_DIS
LIN {X -55.7735,Y -8.9078,Z 71,A -177.5307,B 24.8762,C -2.5678,E1 24.8416,E2 261.3742} C_DIS
LIN {X -56.0619,Y -6.8636,Z 71,A -179.7719,B 24.8758,C -2.572,E1 24.8408,E2 263.619} C_DIS
LIN {X -56.3184,Y -4.2706,Z 71,A 177.5396,B 24.8751,C -2.5795,E1 24.8401,E2 266.3056} C_DIS
LIN {X -56.45,Y -1.8342,Z 71,A 175.0396,B 24.8744,C -2.5869,E1 24.8398,E2 268.803} C_DIS
LIN {X -56.473,Y 0.881,Z 71,A 172.1869,B 24.8737,C -2.594,E1 24.8398,E2 271.6559} C_DIS
LIN {X -56.3544,Y 3.7605,Z 71,A 169.335,B 24.8727,C -2.6044,E1 24.8403,E2 274.5002} C_DIS
LIN {X -56.1354,Y 6.2356,Z 71,A 166.8462,B 24.8718,C -2.6128,E1 24.841,E2 276.9836} C_DIS
LIN {X -55.8067,Y 8.6931,Z 71,A 164.0849,B 24.8714,C -2.6168,E1 24.8421,E2 279.7518} C_DIS
LIN {X -55.2964,Y 11.5015,Z 71,A 161.0004,B 24.8708,C -2.6229,E1 24.8438,E2 282.8401} C_DIS
LIN {X -54.6433,Y 14.287,Z 71,A 158.367,B 24.8695,C -2.6362,E1 24.8455,E2 285.4571} C_DIS
LIN {X -53.839,Y 17.071,Z 71,A 155.3878,B 24.8687,C -2.6445,E1 24.8479,E2 288.4334} C_DIS
LIN {X -52.8868,Y 19.8237,Z 71,A 152.5291,B 24.8676,C -2.6551,E1 24.8506,E2 291.2832} C_DIS
LIN {X -51.9607,Y 22.138,Z 71,A 149.9266,B 24.867,C -2.6614,E1 24.8534,E2 293.8849} C_DIS
LIN {X -50.3651,Y 25.5604,Z 71,A 146.5345,B 24.8651,C -2.6798,E1 24.8574,E2 297.2515} C_DIS
LIN {X -49.3589,Y 27.4529,Z 71,A 142.9999,B 24.8667,C -2.664,E1 24.8623,E2 300.8424} C_DIS
LIN {X -46.951,Y 31.3953,Z 71,A 139.1126,B 24.8641,C -2.6899,E1 24.8681,E2 304.6876} C_DIS
LIN {X -44.9306,Y 34.2241,Z 71,A 135.8446,B 24.8627,C -2.7035,E1 24.8734,E2 307.9389} C_DIS
LIN {X -43.5772,Y 35.9309,Z 71,A 132.7754,B 24.8636,C -2.695,E1 24.8789,E2 311.0426} C_DIS
LIN {X -39.9854,Y 39.8898,Z 71,A 127.5711,B 24.8619,C -2.7118,E1 24.8888,E2 316.2295} C_DIS
LIN {X -37.4639,Y 42.2668,Z 71,A 124.3742,B 24.8605,C -2.7251,E1 24.8954,E2 319.4075} C_DIS
LIN {X -33.5721,Y 45.4195,Z 71,A 119.2662,B 24.8595,C -2.7354,E1 24.9066,E2 324.5099} C_DIS
LIN {X -31.3453,Y 46.9842,Z 71,A 115.9948,B 24.8598,C -2.732,E1 24.9142,E2 327.8003} C_DIS
LIN {X -27.977,Y 49.064,Z 71,A 112.3829,B 24.8584,C -2.7461,E1 24.9228,E2 331.3896} C_DIS
LIN {X -26.115,Y 50.0801,Z 71,A 109.393,B 24.8595,C -2.7351,E1 24.9303,E2 334.4139} C_DIS
LIN {X -23.1774,Y 51.505,Z 71,A 107.0768,B 24.8572,C -2.7574,E1 24.936,E2 336.6827} C_DIS
LIN {X -20.747,Y 52.5312,Z 71,A 104.2864,B 24.857,C -2.759,E1 24.9433,E2 339.4754} C_DIS
LIN {X -18.0633,Y 53.5133,Z 71,A 101.4584,B 24.8565,C -2.7639,E1 24.9507,E2 342.2974} C_DIS
LIN {X -15.5741,Y 54.2903,Z 71,A 98.2973,B 24.8572,C -2.7575,E1 24.9592,E2 345.479} C_DIS
LIN {X -11.9565,Y 55.1996,Z 71,A 94.9388,B 24.856,C -2.7686,E1 24.9683,E2 348.8155} C_DIS
LIN {X -8.7169,Y 55.803,Z 71,A 91.7977,B 24.8554,C -2.7748,E1 24.9769,E2 351.9449} C_DIS
LIN {X -6.2282,Y 56.1362,Z 71,A 89.0896,B 24.8555,C -2.7732,E1 24.9844,E2 354.6586} C_DIS
LIN {X -3.6777,Y 56.36,Z 71,A 86.4789,B 24.8555,C -2.7741,E1 24.9917,E2 357.2683} C_DIS
LIN {X -0.8711,Y 56.4732,Z 71,A 83.6299,B 24.8554,C -2.7749,E1 24.9996,E2 360.1157} C_DIS
LIN {X 1.8314,Y 56.45,Z 71,A 80.9566,B 24.8552,C -2.7766,E1 25.0071,E2 362.7846} C_DIS
LIN {X 4.4304,Y 56.3057,Z 71,A 78.3144,B 24.8552,C -2.7766,E1 25.0144,E2 365.4259} C_DIS
LIN {X 6.881,Y 56.0598,Z 71,A 75.7099,B 24.8554,C -2.7741,E1 25.0217,E2 368.0343} C_DIS
LIN {X 9.6753,Y 55.6457,Z 71,A 72.7277,B 24.8558,C -2.7709,E1 25.0299,E2 371.021} C_DIS
LIN {X 12.7058,Y 55.0319,Z 71,A 69.393,B 24.8563,C -2.7656,E1 25.039,E2 374.3641} C_DIS
LIN {X 16.2491,Y 54.0921,Z 71,A 65.7941,B 24.8563,C -2.7654,E1 25.0487,E2 377.9574} C_DIS
LIN {X 20.0612,Y 52.7968,Z 71,A 62.1311,B 24.8558,C -2.7703,E1 25.0583,E2 381.6013} C_DIS
LIN {X 22.4944,Y 51.807,Z 71,A 59.4412,B 24.8562,C -2.7671,E1 25.0652,E2 384.2926} C_DIS
LIN {X 24.796,Y 50.7465,Z 71,A 56.6534,B 24.857,C -2.7596,E1 25.0723,E2 387.0909} C_DIS
LIN {X 27.343,Y 49.4203,Z 71,A 53.8739,B 24.857,C -2.7586,E1 25.0791,E2 389.865} C_DIS
LIN {X 29.7832,Y 47.989,Z 71,A 50.7928,B 24.858,C -2.75,E1 25.0865,E2 392.9568} C_DIS
LIN {X 32.8032,Y 45.9772,Z 71,A 47.4096,B 24.858,C -2.7503,E1 25.0943,E2 396.328} C_DIS
LIN {X 35.4109,Y 44.0007,Z 71,A 44.453,B 24.8577,C -2.7521,E1 25.1008,E2 399.2694} C_DIS
LIN {X 36.8567,Y 42.7975,Z 71,A 42.0804,B 24.8591,C -2.7386,E1 25.1059,E2 401.6648} C_DIS
LIN {X 38.9362,Y 40.915,Z 71,A 39.2038,B 24.8598,C -2.7323,E1 25.1118,E2 404.5446} C_DIS
LIN {X 40.9307,Y 38.9187,Z 71,A 36.4683,B 24.8601,C -2.7289,E1 25.1171,E2 407.2764} C_DIS
LIN {X 42.8178,Y 36.8314,Z 71,A 33.3233,B 24.8614,C -2.7163,E1 25.1229,E2 410.437} C_DIS
LIN {X 44.5414,Y 34.7278,Z 71,A 30.61,B 24.862,C -2.7108,E1 25.1276,E2 413.1507} C_DIS
LIN {X 46.0436,Y 32.7102,Z 71,A 28.228,B 24.8622,C -2.7083,E1 25.1315,E2 415.5272} C_DIS
LIN {X 47.6301,Y 30.3539,Z 71,A 25.4023,B 24.8629,C -2.7022,E1 25.1359,E2 418.3531} C_DIS
LIN {X 48.9826,Y 28.1186,Z 71,A 22.7922,B 24.8635,C -2.6962,E1 25.1396,E2 420.9641} C_DIS
LIN {X 50.2711,Y 25.7443,Z 71,A 19.6554,B 24.8651,C -2.6801,E1 25.1436,E2 424.1224} C_DIS
LIN {X 51.4587,Y 23.2801,Z 71,A 17.4192,B 24.8647,C -2.6843,E1 25.1463,E2 426.3366} C_DIS
LIN {X 52.4553,Y 20.9401,Z 71,A 14.7984,B 24.8655,C -2.676,E1 25.1491,E2 428.9624} C_DIS
LIN {X 53.3337,Y 18.5873,Z 71,A 12.1864,B 24.8664,C -2.6672,E1 25.1515,E2 431.5806} C_DIS
LIN {X 54.1745,Y 15.9713,Z 71,A 9.4348,B 24.8672,C -2.6598,E1 25.1538,E2 434.3341} C_DIS
LIN {X 54.8642,Y 13.4117,Z 71,A 6.9992,B 24.8674,C -2.6574,E1 25.1555,E2 436.7614} C_DIS
LIN {X 55.553,Y 10.1906,Z 71,A 3.908,B 24.8678,C -2.6529,E1 25.1573,E2 439.8453} C_DIS
LIN {X 56.0363,Y 7.0659,Z 71,A 0.2827,B 24.8698,C -2.6335,E1 25.1587,E2 443.495} C_DIS
LIN {X 56.3402,Y 3.9692,Z 71,A -2.9184,B 24.8709,C -2.6227,E1 25.1595,E2 446.7028} C_DIS
LIN {X 56.464,Y 1.3708,Z 71,A -5.4612,B 24.8715,C -2.6165,E1 25.1598,E2 449.2449} C_DIS
LIN {X 56.4661,Y -1.2551,Z 71,A -8.1737,B 24.8724,C -2.607,E1 25.1597,E2 451.9639} C_DIS
LIN {X 56.3301,Y -4.1191,Z 71,A -11.1807,B 24.8735,C -2.5956,E1 25.1592,E2 454.9799} C_DIS
LIN {X 56.0588,Y -6.8895,Z 71,A -13.8168,B 24.874,C -2.5909,E1 25.1584,E2 457.6116} C_DIS
LIN {X 55.6512,Y -9.644,Z 71,A -16.7081,B 24.875,C -2.5805,E1 25.1571,E2 460.5105} C_DIS
LIN {X 55.0642,Y -12.5663,Z 71,A -19.5906,B 24.8756,C -2.5742,E1 25.1554,E2 463.391} C_DIS
LIN {X 54.3831,Y -15.2464,Z 71,A -22.7314,B 24.8772,C -2.558,E1 25.1531,E2 466.5522} C_DIS
LIN {X 53.4526,Y -18.2433,Z 71,A -25.2882,B 24.8767,C -2.5623,E1 25.1509,E2 469.0843} C_DIS
LIN {X 52.5756,Y -20.6339,Z 71,A -28.3331,B 24.8785,C -2.5441,E1 25.1479,E2 472.1553} C_DIS
LIN {X 51.5329,Y -23.1153,Z 71,A -30.9136,B 24.879,C -2.5393,E1 25.145,E2 474.733} C_DIS
LIN {X 49.9537,Y -26.355,Z 71,A -34.4623,B 24.8797,C -2.531,E1 25.1406,E2 478.2824} C_DIS
LIN {X 48.6455,Y -28.6979,Z 71,A -37.2483,B 24.8806,C -2.5219,E1 25.1367,E2 481.0756} C_DIS
LIN {X 47.2752,Y -30.9039,Z 71,A -40.0704,B 24.8817,C -2.5104,E1 25.1324,E2 483.9107} C_DIS
LIN {X 45.362,Y -33.6489,Z 71,A -43.3801,B 24.8824,C -2.5031,E1 25.127,E2 487.2216} C_DIS
LIN {X 43.7128,Y -35.7661,Z 71,A -45.9368,B 24.8827,C -2.4997,E1 25.1226,E2 489.7745} C_DIS
LIN {X 41.8796,Y -37.8965,Z 71,A -49.539,B 24.8849,C -2.4761,E1 25.1158,E2 493.4164} C_DIS
LIN {X 38.2442,Y -41.5613,Z 71,A -53.6083,B 24.8837,C -2.4892,E1 25.1077,E2 497.4378} C_DIS
LIN {X 37.0917,Y -42.593,Z 71,A -55.5307,B 24.8848,C -2.4779,E1 25.1037,E2 499.3791} C_DIS
LIN {X 34.9502,Y -44.3671,Z 71,A -58.3583,B 24.8853,C -2.4717,E1 25.0975,E2 502.2108} C_DIS
LIN {X 31.7598,Y -46.7042,Z 71,A -62.2101,B 24.8858,C -2.467,E1 25.0888,E2 506.0602} C_DIS
LIN {X 29.67,Y -48.0597,Z 71,A -64.8348,B 24.8864,C -2.4602,E1 25.0826,E2 508.6926} C_DIS
LIN {X 27.3043,Y -49.4419,Z 71,A -67.5449,B 24.8867,C -2.4568,E1 25.076,E2 511.4028} C_DIS
LIN {X 23.7227,Y -51.2562,Z 71,A -71.6557,B 24.8874,C -2.4495,E1 25.0657,E2 515.5199} C_DIS
LIN {X 20.5549,Y -52.6066,Z 71,A -75.1959,B 24.8879,C -2.4435,E1 25.0565,E2 519.0659} C_DIS
LIN {X 17.6863,Y -53.64,Z 71,A -78.2434,B 24.8882,C -2.4406,E1 25.0485,E2 522.1143} C_DIS
LIN {X 15.781,Y -54.2307,Z 71,A -80.5653,B 24.889,C -2.4322,E1 25.0422,E2 524.452} C_DIS
LIN {X 13.3049,Y -54.8903,Z 71,A -82.8998,B 24.8887,C -2.4351,E1 25.0359,E2 526.7764} C_DIS
LIN {X 10.7124,Y -55.4545,Z 71,A -85.3907,B 24.8886,C -2.4368,E1 25.0291,E2 529.2599} C_DIS
LIN {X 8.2675,Y -55.8722,Z 71,A -88.0725,B 24.889,C -2.4317,E1 25.0217,E2 531.9515} C_DIS
LIN {X 5.5427,Y -56.208,Z 71,A -90.4947,B 24.8885,C -2.4373,E1 25.015,E2 534.3585} C_DIS
LIN {X 3.591,Y -56.3658,Z 71,A -92.8736,B 24.8893,C -2.4286,E1 25.0084,E2 536.757} C_DIS
LIN {X 0.6425,Y -56.4768,Z 71,A -95.7395,B 24.8892,C -2.4302,E1 25.0004,E2 539.6186} C_DIS
LIN {X 0.6425,Y -56.4768,Z 71,A -95.7395,B 24.8892,C -2.4302,E1 25.0004,E2 539.6186} C_DIS
Enddeposition()
LIN {X 0.3163,Y -55.5576,Z 71,A -95.8088,B 24.8872,C -2.4513,E1 25.0004,E2 539.6376} C_DIS
Startdeposition()
$VEL.CP = VEL_PRINT
LIN {X 2.0392,Y -55.5243,Z 71,A -93.0503,B 24.8854,C -2.4712,E1 25.0081,E2 536.8326} C_DIS
LIN {X 4.7535,Y -55.358,Z 71,A -90.2485,B 24.8853,C -2.4724,E1 25.0159,E2 534.0291} C_DIS
LIN {X 7.4786,Y -55.0562,Z 71,A -87.4252,B 24.8851,C -2.4741,E1 25.0238,E2 531.204} C_DIS
LIN {X 10.1661,Y -54.6238,Z 71,A -84.6224,B 24.8849,C -2.4761,E1 25.0315,E2 528.3993} C_DIS
LIN {X 12.8297,Y -54.0602,Z 71,A -81.8203,B 24.8847,C -2.4786,E1 25.0391,E2 525.5952} C_DIS
LIN {X 15.4827,Y -53.361,Z 71,A -79.0059,B 24.8844,C -2.4813,E1 25.0467,E2 522.779} C_DIS
LIN {X 18.0421,Y -52.5507,Z 71,A -76.2434,B 24.8841,C -2.4845,E1 25.054,E2 520.0142} C_DIS
LIN {X 20.5351,Y -51.6272,Z 71,A -73.4739,B 24.8837,C -2.4888,E1 25.0613,E2 517.2405} C_DIS
LIN {X 23.1289,Y -50.5189,Z 71,A -70.6051,B 24.8834,C -2.4923,E1 25.0686,E2 514.3705} C_DIS
LIN {X 25.591,Y -49.3175,Z 71,A -67.7906,B 24.883,C -2.4966,E1 25.0756,E2 511.5533} C_DIS
LIN {X 27.9734,Y -48.0062,Z 71,A -64.9957,B 24.8826,C -2.5013,E1 25.0824,E2 508.7555} C_DIS
LIN {X 30.2885,Y -46.5802,Z 71,A -62.2035,B 24.8821,C -2.5064,E1 25.089,E2 505.9605} C_DIS
LIN {X 32.5595,Y -45.0221,Z 71,A -59.3807,B 24.8816,C -2.5117,E1 25.0955,E2 503.1348} C_DIS
LIN {X 34.7176,Y -43.3798,Z 71,A -56.5934,B 24.881,C -2.5174,E1 25.1016,E2 500.3442} C_DIS
LIN {X 36.7928,Y -41.6341,Z 71,A -53.7488,B 24.8803,C -2.5247,E1 25.1076,E2 497.4935} C_DIS
LIN {X 38.7776,Y -39.7919,Z 71,A -50.9811,B 24.8798,C -2.5307,E1 25.1132,E2 494.7231} C_DIS
Enddeposition()
END
